LIN {X 0,Y 429.47,Z 573.716,A -85,B 0,C 180,E1 8276.93,E2 8276.93} C_VEL
LIN {X 0,Y 430.465,Z 577.307,A -85,B 0,C 180,E1 8273.605,E2 8273.605} C_VEL
LIN {X 0,Y 428.623,Z 593.36,A -85,B 0,C 180,E1 8273.398,E2 8273.398} C_VEL
LIN {X 0,Y 427.65,Z 601.061,A -85,B 0,C 180,E1 8273.433,E2 8273.433} C_VEL
LIN {X 0,Y 424.746,Z 621.669,A -85,B 0,C 180,E1 8274.011,E2 8274.011} C_VEL
LIN {X 0,Y 423.922,Z 628.276,A -85,B 0,C 180,E1 8274.029,E2 8274.029} C_VEL
LIN {X 0,Y 413.389,Z 717.354,A -85,B 0,C 180,E1 8272.887,E2 8272.887} C_VEL
LIN {X 0,Y 408.118,Z 746.071,A -85,B 0,C 180,E1 8272.482,E2 8272.482} C_VEL
LIN {X 0,Y 402.723,Z 767.743,A -85,B 0,C 180,E1 8272.122,E2 8272.122} C_VEL
LIN {X 0,Y 395.883,Z 790.196,A -85,B 0,C 180,E1 8271.668,E2 8271.668} C_VEL
LIN {X 0,Y 386.127,Z 816.317,A -85,B 0,C 180,E1 8270.974,E2 8270.974} C_VEL
LIN {X 0,Y 377.346,Z 836.309,A -85,B 0,C 180,E1 8270.305,E2 8270.305} C_VEL
LIN {X 0,Y 367.124,Z 856.797,A -85,B 0,C 180,E1 8269.485,E2 8269.485} C_VEL
LIN {X 0,Y 353.895,Z 879.891,A -85,B 0,C 180,E1 8268.336,E2 8268.336} C_VEL
LIN {X 0,Y 341.958,Z 898.335,A -85,B 0,C 180,E1 8267.201,E2 8267.201} C_VEL
LIN {X 0,Y 329.398,Z 915.934,A -85,B 0,C 180,E1 8265.892,E2 8265.892} C_VEL
LIN {X 0,Y 312.582,Z 937.05,A -85,B 0,C 180,E1 8263.94,E2 8263.94} C_VEL
LIN {X 0,Y 298.439,Z 953.025,A -85,B 0,C 180,E1 8262.084,E2 8262.084} C_VEL
LIN {X 0,Y 284.163,Z 967.885,A -85,B 0,C 180,E1 8259.966,E2 8259.966} C_VEL
LIN {X 0,Y 265.558,Z 985.544,A -85,B 0,C 180,E1 8256.739,E2 8256.739} C_VEL
LIN {X 0,Y 250.897,Z 998.283,A -85,B 0,C 180,E1 8253.725,E2 8253.725} C_VEL
LIN {X 0,Y 235.594,Z 1010.758,A -85,B 0,C 180,E1 8249.974,E2 8249.974} C_VEL
LIN {X 0,Y 218.823,Z 1023.439,A -85,B 0,C 180,E1 8244.877,E2 8244.877} C_VEL
LIN {X 0,Y 206.757,Z 1032.129,A -85,B 0,C 180,E1 8240.258,E2 8240.258} C_VEL
LIN {X 0,Y 194.64,Z 1040.684,A -85,B 0,C 180,E1 8234.318,E2 8234.318} C_VEL
LIN {X 0,Y 183.379,Z 1048.53,A -85,B 0,C 180,E1 8226.723,E2 8226.723} C_VEL
LIN {X 0,Y 176.363,Z 1053.655,A -85,B 0,C 180,E1 8219.838,E2 8219.838} C_VEL
LIN {X 0,Y 171.437,Z 1057.709,A -85,B 0,C 180,E1 8212.278,E2 8212.278} C_VEL
LIN {X 0,Y 168.576,Z 1060.697,A -85,B 0,C 180,E1 8203.375,E2 8203.375} C_VEL
LIN {X 0,Y 167.948,Z 1061.835,A -85,B 0,C 180,E1 8196.495,E2 8196.495} C_VEL
LIN {X 0,Y 167.927,Z 1062.025,A -85,B 0,C 180,E1 8190.341,E2 8190.341} C_VEL
LIN {X 0,Y 167.919,Z 1061.465,A -85,B 0,C 180,E1 8184.533,E2 8184.533} C_VEL
LIN {X 0,Y 168.39,Z 1059.828,A -85,B 0,C 180,E1 8177.657,E2 8177.657} C_VEL
LIN {X 0,Y 170.075,Z 1057.173,A -85,B 0,C 180,E1 8170.778,E2 8170.778} C_VEL
LIN {X 0,Y 173.594,Z 1053.274,A -85,B 0,C 180,E1 8163.672,E2 8163.672} C_VEL
LIN {X 0,Y 180.092,Z 1047.442,A -85,B 0,C 180,E1 8155.892,E2 8155.892} C_VEL
LIN {X 0,Y 189.636,Z 1039.498,A -85,B 0,C 180,E1 8148.367,E2 8148.367} C_VEL
LIN {X 0,Y 199.716,Z 1031.446,A -85,B 0,C 180,E1 8142.612,E2 8142.612} C_VEL
LIN {X 0,Y 213.267,Z 1020.629,A -85,B 0,C 180,E1 8136.706,E2 8136.706} C_VEL
LIN {X 0,Y 227.999,Z 1008.192,A -85,B 0,C 180,E1 8131.703,E2 8131.703} C_VEL
LIN {X 0,Y 241.285,Z 996.496,A -85,B 0,C 180,E1 8128.034,E2 8128.034} C_VEL
LIN {X 0,Y 258.503,Z 980.275,A -85,B 0,C 180,E1 8124.099,E2 8124.099} C_VEL
LIN {X 0,Y 272.707,Z 965.724,A -85,B 0,C 180,E1 8121.363,E2 8121.363} C_VEL
LIN {X 0,Y 286.634,Z 950.38,A -85,B 0,C 180,E1 8119.03,E2 8119.03} C_VEL
LIN {X 0,Y 303.56,Z 929.827,A -85,B 0,C 180,E1 8116.562,E2 8116.562} C_VEL
LIN {X 0,Y 316.203,Z 912.825,A -85,B 0,C 180,E1 8114.931,E2 8114.931} C_VEL
LIN {X 0,Y 328.971,Z 893.994,A -85,B 0,C 180,E1 8113.44,E2 8113.44} C_VEL
LIN {X 0,Y 342.461,Z 871.569,A -85,B 0,C 180,E1 8112.014,E2 8112.014} C_VEL
LIN {X 0,Y 352.942,Z 851.881,A -85,B 0,C 180,E1 8110.999,E2 8110.999} C_VEL
LIN {X 0,Y 362.609,Z 831.453,A -85,B 0,C 180,E1 8110.129,E2 8110.129} C_VEL
LIN {X 0,Y 372.867,Z 806.091,A -85,B 0,C 180,E1 8109.259,E2 8109.259} C_VEL
LIN {X 0,Y 380.057,Z 784.957,A -85,B 0,C 180,E1 8108.678,E2 8108.678} C_VEL
LIN {X 0,Y 386.562,Z 762.237,A -85,B 0,C 180,E1 8108.193,E2 8108.193} C_VEL
LIN {X 0,Y 392.552,Z 734.98,A -85,B 0,C 180,E1 8107.729,E2 8107.729} C_VEL
LIN {X 0,Y 396.079,Z 712.548,A -85,B 0,C 180,E1 8107.4,E2 8107.4} C_VEL
LIN {X 0,Y 412.103,Z 569.364,A -85,B 0,C 180,E1 8105.465,E2 8105.465} C_VEL
LIN {X 0,Y 410.53,Z 565.385,A -85,B 0,C 180,E1 8102.513,E2 8102.513} C_VEL
LIN {X 0,Y 409.758,Z 563.185,A -85,B 0,C 180,E1 8098.182,E2 8098.182} C_VEL
LIN {X 0,Y 410.752,Z 565.908,A -85,B 0,C 180,E1 8093.781,E2 8093.781} C_VEL
LIN {X 0,Y 412.109,Z 569.371,A -85,B 0,C 180,E1 8091.348,E2 8091.348} C_VEL
LIN {X 0,Y 395.646,Z 715.398,A -85,B 0,C 180,E1 8089.405,E2 8089.405} C_VEL
LIN {X 0,Y 390.904,Z 742.775,A -85,B 0,C 180,E1 8088.992,E2 8088.992} C_VEL
LIN {X 0,Y 385.342,Z 765.972,A -85,B 0,C 180,E1 8088.555,E2 8088.555} C_VEL
LIN {X 0,Y 379.395,Z 786.292,A -85,B 0,C 180,E1 8088.074,E2 8088.074} C_VEL
LIN {X 0,Y 370.48,Z 811.64,A -85,B 0,C 180,E1 8087.329,E2 8087.329} C_VEL
LIN {X 0,Y 361.399,Z 833.181,A -85,B 0,C 180,E1 8086.531,E2 8086.531} C_VEL
LIN {X 0,Y 351.957,Z 852.896,A -85,B 0,C 180,E1 8085.64,E2 8085.64} C_VEL
LIN {X 0,Y 339.939,Z 875.096,A -85,B 0,C 180,E1 8084.428,E2 8084.428} C_VEL
LIN {X 0,Y 326.959,Z 895.939,A -85,B 0,C 180,E1 8083.014,E2 8083.014} C_VEL
LIN {X 0,Y 314.662,Z 913.816,A -85,B 0,C 180,E1 8081.536,E2 8081.536} C_VEL
LIN {X 0,Y 299.012,Z 934.324,A -85,B 0,C 180,E1 8079.44,E2 8079.44} C_VEL
LIN {X 0,Y 284.739,Z 951.124,A -85,B 0,C 180,E1 8077.277,E2 8077.277} C_VEL
LIN {X 0,Y 270.645,Z 966.445,A -85,B 0,C 180,E1 8074.842,E2 8074.842} C_VEL
LIN {X 0,Y 253.828,Z 983.189,A -85,B 0,C 180,E1 8071.455,E2 8071.455} C_VEL
LIN {X 0,Y 240.068,Z 995.842,A -85,B 0,C 180,E1 8068.175,E2 8068.175} C_VEL
LIN {X 0,Y 226.493,Z 1007.65,A -85,B 0,C 180,E1 8064.32,E2 8064.32} C_VEL
LIN {X 0,Y 210.608,Z 1020.673,A -85,B 0,C 180,E1 8058.706,E2 8058.706} C_VEL
LIN {X 0,Y 199.578,Z 1029.377,A -85,B 0,C 180,E1 8053.739,E2 8053.739} C_VEL
LIN {X 0,Y 189.309,Z 1037.47,A -85,B 0,C 180,E1 8047.784,E2 8047.784} C_VEL
LIN {X 0,Y 179.397,Z 1045.474,A -85,B 0,C 180,E1 8039.739,E2 8039.739} C_VEL
LIN {X 0,Y 173.677,Z 1050.54,A -85,B 0,C 180,E1 8032.689,E2 8032.689} C_VEL
LIN {X 0,Y 170.113,Z 1054.357,A -85,B 0,C 180,E1 8025.428,E2 8025.428} C_VEL
LIN {X 0,Y 168.256,Z 1057.297,A -85,B 0,C 180,E1 8017.053,E2 8017.053} C_VEL
LIN {X 0,Y 167.946,Z 1058.534,A -85,B 0,C 180,E1 8010,E2 8010} C_VEL
LIN {X 0,Y 167.942,Z 1058.789,A -85,B 0,C 180,E1 8003.505,E2 8003.505} C_VEL
LIN {X 0,Y 168.271,Z 1058.165,A -85,B 0,C 180,E1 7996.95,E2 7996.95} C_VEL
LIN {X 0,Y 169.687,Z 1056.537,A -85,B 0,C 180,E1 7990.015,E2 7990.015} C_VEL
LIN {X 0,Y 172.725,Z 1053.867,A -85,B 0,C 180,E1 7983.062,E2 7983.062} C_VEL
LIN {X 0,Y 178.106,Z 1049.841,A -85,B 0,C 180,E1 7975.847,E2 7975.847} C_VEL
LIN {X 0,Y 187.876,Z 1043.071,A -85,B 0,C 180,E1 7967.476,E2 7967.476} C_VEL
LIN {X 0,Y 198.241,Z 1035.985,A -85,B 0,C 180,E1 7961.277,E2 7961.277} C_VEL
LIN {X 0,Y 210.239,Z 1027.705,A -85,B 0,C 180,E1 7955.802,E2 7955.802} C_VEL
LIN {X 0,Y 226.504,Z 1015.937,A -85,B 0,C 180,E1 7950.091,E2 7950.091} C_VEL
LIN {X 0,Y 240.664,Z 1005.04,A -85,B 0,C 180,E1 7946.13,E2 7946.13} C_VEL
LIN {X 0,Y 257.231,Z 991.501,A -85,B 0,C 180,E1 7942.312,E2 7942.312} C_VEL
LIN {X 0,Y 274.025,Z 976.349,A -85,B 0,C 180,E1 7939.081,E2 7939.081} C_VEL
LIN {X 0,Y 288.312,Z 962.437,A -85,B 0,C 180,E1 7936.729,E2 7936.729} C_VEL
LIN {X 0,Y 304.537,Z 945.307,A -85,B 0,C 180,E1 7934.402,E2 7934.402} C_VEL
LIN {X 0,Y 320.435,Z 926.444,A -85,B 0,C 180,E1 7932.397,E2 7932.397} C_VEL
LIN {X 0,Y 333.051,Z 910.04,A -85,B 0,C 180,E1 7930.973,E2 7930.973} C_VEL
LIN {X 0,Y 347.241,Z 889.716,A -85,B 0,C 180,E1 7929.519,E2 7929.519} C_VEL
LIN {X 0,Y 360.273,Z 868.328,A -85,B 0,C 180,E1 7928.298,E2 7928.298} C_VEL
LIN {X 0,Y 370.553,Z 849.453,A -85,B 0,C 180,E1 7927.411,E2 7927.411} C_VEL
LIN {X 0,Y 381.435,Z 826.896,A -85,B 0,C 180,E1 7926.535,E2 7926.535} C_VEL
LIN {X 0,Y 390.957,Z 803.368,A -85,B 0,C 180,E1 7925.801,E2 7925.801} C_VEL
LIN {X 0,Y 398.14,Z 782.602,A -85,B 0,C 180,E1 7925.274,E2 7925.274} C_VEL
LIN {X 0,Y 405.183,Z 758.262,A -85,B 0,C 180,E1 7924.791,E2 7924.791} C_VEL
LIN {X 0,Y 410.782,Z 732.473,A -85,B 0,C 180,E1 7924.388,E2 7924.388} C_VEL
LIN {X 0,Y 414.333,Z 710.195,A -85,B 0,C 180,E1 7924.084,E2 7924.084} C_VEL
LIN {X 0,Y 429.028,Z 584.149,A -85,B 0,C 180,E1 7922.471,E2 7922.471} C_VEL
LIN {X 0,Y 428.424,Z 581.286,A -85,B 0,C 180,E1 7919.465,E2 7919.465} C_VEL
LIN {X 0,Y 428.475,Z 581.6,A -85,B 0,C 180,E1 7917.057,E2 7917.057} C_VEL
LIN {X 0,Y 429.022,Z 584.37,A -85,B 0,C 180,E1 7914.582,E2 7914.582} C_VEL
LIN {X 0,Y 423.922,Z 628.276,A -85,B 0,C 180,E1 7914.029,E2 7914.029} C_VEL
LIN {X 0,Y 422.951,Z 635.978,A -85,B 0,C 180,E1 7914.066,E2 7914.066} C_VEL
LIN {X 0,Y 420.093,Z 656.581,A -85,B 0,C 180,E1 7914.66,E2 7914.66} C_VEL
LIN {X 0,Y 419.271,Z 663.188,A -85,B 0,C 180,E1 7914.678,E2 7914.678} C_VEL
LIN {X 0,Y 412.391,Z 719.368,A -85,B 0,C 180,E1 7913.97,E2 7913.97} C_VEL
LIN {X 0,Y 407.213,Z 746.607,A -85,B 0,C 180,E1 7913.596,E2 7913.596} C_VEL
LIN {X 0,Y 401.82,Z 767.987,A -85,B 0,C 180,E1 7913.256,E2 7913.256} C_VEL
LIN {X 0,Y 394.567,Z 791.474,A -85,B 0,C 180,E1 7912.799,E2 7912.799} C_VEL
LIN {X 0,Y 384.928,Z 816.769,A -85,B 0,C 180,E1 7912.15,E2 7912.15} C_VEL
LIN {X 0,Y 376.077,Z 836.652,A -85,B 0,C 180,E1 7911.512,E2 7911.512} C_VEL
LIN {X 0,Y 365.319,Z 857.898,A -85,B 0,C 180,E1 7910.692,E2 7910.692} C_VEL
LIN {X 0,Y 351.768,Z 881.033,A -85,B 0,C 180,E1 7909.574,E2 7909.574} C_VEL
LIN {X 0,Y 339.795,Z 899.198,A -85,B 0,C 180,E1 7908.49,E2 7908.49} C_VEL
LIN {X 0,Y 325.704,Z 918.528,A -85,B 0,C 180,E1 7907.084,E2 7907.084} C_VEL
LIN {X 0,Y 309.606,Z 938.108,A -85,B 0,C 180,E1 7905.295,E2 7905.295} C_VEL
LIN {X 0,Y 296.015,Z 953.141,A -85,B 0,C 180,E1 7903.597,E2 7903.597} C_VEL
LIN {X 0,Y 280.605,Z 968.825,A -85,B 0,C 180,E1 7901.413,E2 7901.413} C_VEL
LIN {X 0,Y 262.401,Z 985.613,A -85,B 0,C 180,E1 7898.398,E2 7898.398} C_VEL
LIN {X 0,Y 247.337,Z 998.337,A -85,B 0,C 180,E1 7895.448,E2 7895.448} C_VEL
LIN {X 0,Y 230.823,Z 1011.369,A -85,B 0,C 180,E1 7891.565,E2 7891.565} C_VEL
LIN {X 0,Y 214.145,Z 1023.454,A -85,B 0,C 180,E1 7886.698,E2 7886.698} C_VEL
LIN {X 0,Y 201.29,Z 1032.299,A -85,B 0,C 180,E1 7881.978,E2 7881.978} C_VEL
LIN {X 0,Y 187.765,Z 1041.384,A -85,B 0,C 180,E1 7875.527,E2 7875.527} C_VEL
LIN {X 0,Y 176.383,Z 1048.771,A -85,B 0,C 180,E1 7868.003,E2 7868.003} C_VEL
LIN {X 0,Y 169.025,Z 1053.775,A -85,B 0,C 180,E1 7860.975,E2 7860.975} C_VEL
LIN {X 0,Y 163.349,Z 1058.145,A -85,B 0,C 180,E1 7852.304,E2 7852.304} C_VEL
LIN {X 0,Y 160.616,Z 1060.701,A -85,B 0,C 180,E1 7843.684,E2 7843.684} C_VEL
LIN {X 0,Y 159.96,Z 1061.761,A -85,B 0,C 180,E1 7836.821,E2 7836.821} C_VEL
LIN {X 0,Y 159.919,Z 1061.965,A -85,B 0,C 180,E1 7830.717,E2 7830.717} C_VEL
LIN {X 0,Y 159.918,Z 1061.442,A -85,B 0,C 180,E1 7824.619,E2 7824.619} C_VEL
LIN {X 0,Y 160.417,Z 1059.841,A -85,B 0,C 180,E1 7817.399,E2 7817.399} C_VEL
LIN {X 0,Y 162.361,Z 1057.061,A -85,B 0,C 180,E1 7809.826,E2 7809.826} C_VEL
LIN {X 0,Y 166.24,Z 1053.152,A -85,B 0,C 180,E1 7802.411,E2 7802.411} C_VEL
LIN {X 0,Y 173.632,Z 1047.046,A -85,B 0,C 180,E1 7794.029,E2 7794.029} C_VEL
LIN {X 0,Y 183.953,Z 1038.984,A -85,B 0,C 180,E1 7786.345,E2 7786.345} C_VEL
LIN {X 0,Y 194.712,Z 1030.869,A -85,B 0,C 180,E1 7780.535,E2 7780.535} C_VEL
LIN {X 0,Y 209.647,Z 1019.395,A -85,B 0,C 180,E1 7774.401,E2 7774.401} C_VEL
LIN {X 0,Y 223.722,Z 1007.99,A -85,B 0,C 180,E1 7769.883,E2 7769.883} C_VEL
LIN {X 0,Y 238.228,Z 995.638,A -85,B 0,C 180,E1 7766.078,E2 7766.078} C_VEL
LIN {X 0,Y 256.005,Z 979.251,A -85,B 0,C 180,E1 7762.233,E2 7762.233} C_VEL
LIN {X 0,Y 269.87,Z 965.379,A -85,B 0,C 180,E1 7759.704,E2 7759.704} C_VEL
LIN {X 0,Y 284.039,Z 950.103,A -85,B 0,C 180,E1 7757.45,E2 7757.45} C_VEL
LIN {X 0,Y 300.811,Z 930.15,A -85,B 0,C 180,E1 7755.12,E2 7755.12} C_VEL
LIN {X 0,Y 313.679,Z 913.18,A -85,B 0,C 180,E1 7753.538,E2 7753.538} C_VEL
LIN {X 0,Y 326.253,Z 894.982,A -85,B 0,C 180,E1 7752.135,E2 7752.135} C_VEL
LIN {X 0,Y 340.851,Z 871.148,A -85,B 0,C 180,E1 7750.667,E2 7750.667} C_VEL
LIN {X 0,Y 351.011,Z 852.333,A -85,B 0,C 180,E1 7749.732,E2 7749.732} C_VEL
LIN {X 0,Y 360.329,Z 832.982,A -85,B 0,C 180,E1 7748.933,E2 7748.933} C_VEL
LIN {X 0,Y 370.654,Z 808.205,A -85,B 0,C 180,E1 7748.099,E2 7748.099} C_VEL
LIN {X 0,Y 378.444,Z 785.754,A -85,B 0,C 180,E1 7747.5,E2 7747.5} C_VEL
LIN {X 0,Y 384.802,Z 763.973,A -85,B 0,C 180,E1 7747.05,E2 7747.05} C_VEL
LIN {X 0,Y 391.137,Z 736.073,A -85,B 0,C 180,E1 7746.587,E2 7746.587} C_VEL
LIN {X 0,Y 394.832,Z 713.123,A -85,B 0,C 180,E1 7746.258,E2 7746.258} C_VEL
LIN {X 0,Y 410.46,Z 575.932,A -85,B 0,C 180,E1 7744.453,E2 7744.453} C_VEL
LIN {X 0,Y 409.492,Z 573.267,A -85,B 0,C 180,E1 7742.379,E2 7742.379} C_VEL
LIN {X 0,Y 408.781,Z 571.142,A -85,B 0,C 180,E1 7738.178,E2 7738.178} C_VEL
LIN {X 0,Y 409.707,Z 573.818,A -85,B 0,C 180,E1 7733.906,E2 7733.906} C_VEL
LIN {X 0,Y 410.429,Z 576.164,A -85,B 0,C 180,E1 7732.37,E2 7732.37} C_VEL
LIN {X 0,Y 394.459,Z 715.538,A -85,B 0,C 180,E1 7730.554,E2 7730.554} C_VEL
LIN {X 0,Y 389.648,Z 742.945,A -85,B 0,C 180,E1 7730.153,E2 7730.153} C_VEL
LIN {X 0,Y 384.031,Z 766.109,A -85,B 0,C 180,E1 7729.733,E2 7729.733} C_VEL
LIN {X 0,Y 378.06,Z 786.281,A -85,B 0,C 180,E1 7729.275,E2 7729.275} C_VEL
LIN {X 0,Y 369.271,Z 811.091,A -85,B 0,C 180,E1 7728.578,E2 7728.578} C_VEL
LIN {X 0,Y 359.619,Z 833.698,A -85,B 0,C 180,E1 7727.771,E2 7727.771} C_VEL
LIN {X 0,Y 350.054,Z 853.368,A -85,B 0,C 180,E1 7726.911,E2 7726.911} C_VEL
LIN {X 0,Y 337.418,Z 876.224,A -85,B 0,C 180,E1 7725.698,E2 7725.698} C_VEL
LIN {X 0,Y 324.93,Z 895.957,A -85,B 0,C 180,E1 7724.401,E2 7724.401} C_VEL
LIN {X 0,Y 312.63,Z 913.561,A -85,B 0,C 180,E1 7722.997,E2 7722.997} C_VEL
LIN {X 0,Y 297.114,Z 933.624,A -85,B 0,C 180,E1 7721.024,E2 7721.024} C_VEL
LIN {X 0,Y 282.804,Z 950.19,A -85,B 0,C 180,E1 7718.971,E2 7718.971} C_VEL
LIN {X 0,Y 268.893,Z 965.042,A -85,B 0,C 180,E1 7716.704,E2 7716.704} C_VEL
LIN {X 0,Y 252.334,Z 981.35,A -85,B 0,C 180,E1 7713.577,E2 7713.577} C_VEL
LIN {X 0,Y 236.579,Z 995.438,A -85,B 0,C 180,E1 7710.045,E2 7710.045} C_VEL
LIN {X 0,Y 223.168,Z 1006.728,A -85,B 0,C 180,E1 7706.445,E2 7706.445} C_VEL
LIN {X 0,Y 207.578,Z 1019.163,A -85,B 0,C 180,E1 7701.291,E2 7701.291} C_VEL
LIN {X 0,Y 194.274,Z 1029.15,A -85,B 0,C 180,E1 7695.676,E2 7695.676} C_VEL
LIN {X 0,Y 183.355,Z 1037.283,A -85,B 0,C 180,E1 7689.645,E2 7689.645} C_VEL
LIN {X 0,Y 172.691,Z 1045.361,A -85,B 0,C 180,E1 7681.406,E2 7681.406} C_VEL
LIN {X 0,Y 166.346,Z 1050.539,A -85,B 0,C 180,E1 7673.984,E2 7673.984} C_VEL
LIN {X 0,Y 162.43,Z 1054.356,A -85,B 0,C 180,E1 7666.449,E2 7666.449} C_VEL
LIN {X 0,Y 160.346,Z 1057.294,A -85,B 0,C 180,E1 7657.885,E2 7657.885} C_VEL
LIN {X 0,Y 159.951,Z 1058.594,A -85,B 0,C 180,E1 7650.358,E2 7650.358} C_VEL
LIN {X 0,Y 159.939,Z 1058.896,A -85,B 0,C 180,E1 7643.735,E2 7643.735} C_VEL
LIN {X 0,Y 160.298,Z 1058.296,A -85,B 0,C 180,E1 7636.656,E2 7636.656} C_VEL
LIN {X 0,Y 161.961,Z 1056.591,A -85,B 0,C 180,E1 7629.018,E2 7629.018} C_VEL
LIN {X 0,Y 165.3,Z 1053.952,A -85,B 0,C 180,E1 7621.848,E2 7621.848} C_VEL
LIN {X 0,Y 170.916,Z 1050.08,A -85,B 0,C 180,E1 7614.608,E2 7614.608} C_VEL
LIN {X 0,Y 180.863,Z 1043.688,A -85,B 0,C 180,E1 7606.287,E2 7606.287} C_VEL
LIN {X 0,Y 192.233,Z 1036.337,A -85,B 0,C 180,E1 7599.663,E2 7599.663} C_VEL
LIN {X 0,Y 204.649,Z 1028.189,A -85,B 0,C 180,E1 7594.186,E2 7594.186} C_VEL
LIN {X 0,Y 221.691,Z 1016.415,A -85,B 0,C 180,E1 7588.418,E2 7588.418} C_VEL
LIN {X 0,Y 236.248,Z 1005.617,A -85,B 0,C 180,E1 7584.501,E2 7584.501} C_VEL
LIN {X 0,Y 250.963,Z 993.989,A -85,B 0,C 180,E1 7581.204,E2 7581.204} C_VEL
LIN {X 0,Y 269.727,Z 977.804,A -85,B 0,C 180,E1 7577.692,E2 7577.692} C_VEL
LIN {X 0,Y 284.17,Z 964.146,A -85,B 0,C 180,E1 7575.399,E2 7575.399} C_VEL
LIN {X 0,Y 299.025,Z 948.913,A -85,B 0,C 180,E1 7573.332,E2 7573.332} C_VEL
LIN {X 0,Y 316.3,Z 929.304,A -85,B 0,C 180,E1 7571.221,E2 7571.221} C_VEL
LIN {X 0,Y 329.734,Z 912.297,A -85,B 0,C 180,E1 7569.759,E2 7569.759} C_VEL
LIN {X 0,Y 342.234,Z 894.891,A -85,B 0,C 180,E1 7568.516,E2 7568.516} C_VEL
LIN {X 0,Y 356.78,Z 872.204,A -85,B 0,C 180,E1 7567.209,E2 7567.209} C_VEL
LIN {X 0,Y 368.158,Z 851.855,A -85,B 0,C 180,E1 7566.267,E2 7566.267} C_VEL
LIN {X 0,Y 377.711,Z 832.613,A -85,B 0,C 180,E1 7565.524,E2 7565.524} C_VEL
LIN {X 0,Y 388.288,Z 808.07,A -85,B 0,C 180,E1 7564.749,E2 7564.749} C_VEL
LIN {X 0,Y 396.506,Z 785.025,A -85,B 0,C 180,E1 7564.175,E2 7564.175} C_VEL
LIN {X 0,Y 402.699,Z 764.375,A -85,B 0,C 180,E1 7563.767,E2 7563.767} C_VEL
LIN {X 0,Y 408.913,Z 738.596,A -85,B 0,C 180,E1 7563.356,E2 7563.356} C_VEL
LIN {X 0,Y 413.167,Z 713.559,A -85,B 0,C 180,E1 7563.021,E2 7563.021} C_VEL
LIN {X 0,Y 427.715,Z 591.178,A -85,B 0,C 180,E1 7561.474,E2 7561.474} C_VEL
LIN {X 0,Y 427.448,Z 589.227,A -85,B 0,C 180,E1 7559.464,E2 7559.464} C_VEL
LIN {X 0,Y 427.485,Z 589.541,A -85,B 0,C 180,E1 7557.135,E2 7557.135} C_VEL
LIN {X 0,Y 427.714,Z 591.357,A -85,B 0,C 180,E1 7555.567,E2 7555.567} C_VEL
LIN {X 0,Y 419.271,Z 663.188,A -85,B 0,C 180,E1 7554.678,E2 7554.678} C_VEL
LIN {X 0,Y 418.304,Z 670.889,A -85,B 0,C 180,E1 7554.717,E2 7554.717} C_VEL
LIN {X 0,Y 415.494,Z 691.484,A -85,B 0,C 180,E1 7555.328,E2 7555.328} C_VEL
LIN {X 0,Y 414.674,Z 698.09,A -85,B 0,C 180,E1 7555.348,E2 7555.348} C_VEL
LIN {X 0,Y 410.27,Z 728.43,A -85,B 0,C 180,E1 7554.967,E2 7554.967} C_VEL
LIN {X 0,Y 405.642,Z 750.656,A -85,B 0,C 180,E1 7554.667,E2 7554.667} C_VEL
LIN {X 0,Y 399.101,Z 775.285,A -85,B 0,C 180,E1 7554.274,E2 7554.274} C_VEL
LIN {X 0,Y 390.762,Z 799.859,A -85,B 0,C 180,E1 7553.771,E2 7553.771} C_VEL
LIN {X 0,Y 382.541,Z 820.389,A -85,B 0,C 180,E1 7553.245,E2 7553.245} C_VEL
LIN {X 0,Y 371.547,Z 844.159,A -85,B 0,C 180,E1 7552.483,E2 7552.483} C_VEL
LIN {X 0,Y 359.498,Z 866.24,A -85,B 0,C 180,E1 7551.592,E2 7551.592} C_VEL
LIN {X 0,Y 348.522,Z 884.184,A -85,B 0,C 180,E1 7550.72,E2 7550.72} C_VEL
LIN {X 0,Y 334.103,Z 905.369,A -85,B 0,C 180,E1 7549.457,E2 7549.457} C_VEL
LIN {X 0,Y 318.639,Z 925.256,A -85,B 0,C 180,E1 7547.956,E2 7547.956} C_VEL
LIN {X 0,Y 304.935,Z 941.267,A -85,B 0,C 180,E1 7546.465,E2 7546.465} C_VEL
LIN {X 0,Y 288.531,Z 958.784,A -85,B 0,C 180,E1 7544.448,E2 7544.448} C_VEL
LIN {X 0,Y 271.243,Z 975.26,A -85,B 0,C 180,E1 7542.002,E2 7542.002} C_VEL
LIN {X 0,Y 256.167,Z 988.472,A -85,B 0,C 180,E1 7539.518,E2 7539.518} C_VEL
LIN {X 0,Y 238.49,Z 1002.819,A -85,B 0,C 180,E1 7536.061,E2 7536.061} C_VEL
LIN {X 0,Y 221.05,Z 1015.595,A -85,B 0,C 180,E1 7531.891,E2 7531.891} C_VEL
LIN {X 0,Y 206.959,Z 1025.303,A -85,B 0,C 180,E1 7527.724,E2 7527.724} C_VEL
LIN {X 0,Y 191.052,Z 1035.72,A -85,B 0,C 180,E1 7521.724,E2 7521.724} C_VEL
LIN {X 0,Y 177.894,Z 1043.82,A -85,B 0,C 180,E1 7515.089,E2 7515.089} C_VEL
LIN {X 0,Y 168.032,Z 1049.921,A -85,B 0,C 180,E1 7508.233,E2 7508.233} C_VEL
LIN {X 0,Y 159.124,Z 1055.678,A -85,B 0,C 180,E1 7498.937,E2 7498.937} C_VEL
LIN {X 0,Y 154.472,Z 1059.035,A -85,B 0,C 180,E1 7490.459,E2 7490.459} C_VEL
LIN {X 0,Y 152.467,Z 1060.914,A -85,B 0,C 180,E1 7482.884,E2 7482.884} C_VEL
LIN {X 0,Y 151.944,Z 1061.735,A -85,B 0,C 180,E1 7476.423,E2 7476.423} C_VEL
LIN {X 0,Y 151.926,Z 1061.86,A -85,B 0,C 180,E1 7470.377,E2 7470.377} C_VEL
LIN {X 0,Y 151.932,Z 1061.281,A -85,B 0,C 180,E1 7463.956,E2 7463.956} C_VEL
LIN {X 0,Y 152.568,Z 1059.624,A -85,B 0,C 180,E1 7456.354,E2 7456.354} C_VEL
LIN {X 0,Y 154.693,Z 1056.949,A -85,B 0,C 180,E1 7448.779,E2 7448.779} C_VEL
LIN {X 0,Y 158.966,Z 1053.029,A -85,B 0,C 180,E1 7441.032,E2 7441.032} C_VEL
LIN {X 0,Y 166.981,Z 1046.908,A -85,B 0,C 180,E1 7432.354,E2 7432.354} C_VEL
LIN {X 0,Y 177.634,Z 1039.103,A -85,B 0,C 180,E1 7424.718,E2 7424.718} C_VEL
LIN {X 0,Y 188.806,Z 1031.113,A -85,B 0,C 180,E1 7418.878,E2 7418.878} C_VEL
LIN {X 0,Y 203.714,Z 1020.249,A -85,B 0,C 180,E1 7412.932,E2 7412.932} C_VEL
LIN {X 0,Y 218.955,Z 1008.369,A -85,B 0,C 180,E1 7408.194,E2 7408.194} C_VEL
LIN {X 0,Y 233.284,Z 996.587,A -85,B 0,C 180,E1 7404.567,E2 7404.567} C_VEL
LIN {X 0,Y 250.533,Z 981.346,A -85,B 0,C 180,E1 7400.949,E2 7400.949} C_VEL
LIN {X 0,Y 266.412,Z 965.899,A -85,B 0,C 180,E1 7398.151,E2 7398.151} C_VEL
LIN {X 0,Y 279.93,Z 951.698,A -85,B 0,C 180,E1 7396.087,E2 7396.087} C_VEL
LIN {X 0,Y 296.158,Z 933.126,A -85,B 0,C 180,E1 7393.916,E2 7393.916} C_VEL
LIN {X 0,Y 310.948,Z 914.072,A -85,B 0,C 180,E1 7392.166,E2 7392.166} C_VEL
LIN {X 0,Y 323.201,Z 896.712,A -85,B 0,C 180,E1 7390.86,E2 7390.86} C_VEL
LIN {X 0,Y 337.106,Z 874.825,A -85,B 0,C 180,E1 7389.522,E2 7389.522} C_VEL
LIN {X 0,Y 349.252,Z 852.784,A -85,B 0,C 180,E1 7388.452,E2 7388.452} C_VEL
LIN {X 0,Y 358.607,Z 833.652,A -85,B 0,C 180,E1 7387.691,E2 7387.691} C_VEL
LIN {X 0,Y 368.644,Z 810.182,A -85,B 0,C 180,E1 7386.923,E2 7386.923} C_VEL
LIN {X 0,Y 376.95,Z 786.68,A -85,B 0,C 180,E1 7386.316,E2 7386.316} C_VEL
LIN {X 0,Y 383.291,Z 765.353,A -85,B 0,C 180,E1 7385.89,E2 7385.89} C_VEL
LIN {X 0,Y 389.416,Z 739.696,A -85,B 0,C 180,E1 7385.472,E2 7385.472} C_VEL
LIN {X 0,Y 393.635,Z 714.463,A -85,B 0,C 180,E1 7385.12,E2 7385.12} C_VEL
LIN {X 0,Y 408.929,Z 582.638,A -85,B 0,C 180,E1 7383.434,E2 7383.434} C_VEL
LIN {X 0,Y 408.402,Z 581.066,A -85,B 0,C 180,E1 7382.105,E2 7382.105} C_VEL
LIN {X 0,Y 407.803,Z 579.102,A -85,B 0,C 180,E1 7378.173,E2 7378.173} C_VEL
LIN {X 0,Y 408.638,Z 581.623,A -85,B 0,C 180,E1 7374.101,E2 7374.101} C_VEL
LIN {X 0,Y 408.894,Z 582.831,A -85,B 0,C 180,E1 7373.402,E2 7373.402} C_VEL
LIN {X 0,Y 393.425,Z 715.701,A -85,B 0,C 180,E1 7371.709,E2 7371.709} C_VEL
LIN {X 0,Y 388.5,Z 743.337,A -85,B 0,C 180,E1 7371.318,E2 7371.318} C_VEL
LIN {X 0,Y 382.85,Z 766.362,A -85,B 0,C 180,E1 7370.917,E2 7370.917} C_VEL
LIN {X 0,Y 376.658,Z 787.001,A -85,B 0,C 180,E1 7370.466,E2 7370.466} C_VEL
LIN {X 0,Y 367.306,Z 812.781,A -85,B 0,C 180,E1 7369.762,E2 7369.762} C_VEL
LIN {X 0,Y 358.01,Z 834.214,A -85,B 0,C 180,E1 7369.022,E2 7369.022} C_VEL
LIN {X 0,Y 348.326,Z 853.839,A -85,B 0,C 180,E1 7368.196,E2 7368.196} C_VEL
LIN {X 0,Y 335.066,Z 877.352,A -85,B 0,C 180,E1 7366.987,E2 7366.987} C_VEL
LIN {X 0,Y 322.854,Z 896.329,A -85,B 0,C 180,E1 7365.781,E2 7365.781} C_VEL
LIN {X 0,Y 310.363,Z 913.908,A -85,B 0,C 180,E1 7364.424,E2 7364.424} C_VEL
LIN {X 0,Y 294.142,Z 934.428,A -85,B 0,C 180,E1 7362.46,E2 7362.46} C_VEL
LIN {X 0,Y 279.142,Z 951.39,A -85,B 0,C 180,E1 7360.401,E2 7360.401} C_VEL
LIN {X 0,Y 264.953,Z 966.144,A -85,B 0,C 180,E1 7358.18,E2 7358.18} C_VEL
LIN {X 0,Y 246.31,Z 983.773,A -85,B 0,C 180,E1 7354.77,E2 7354.77} C_VEL
LIN {X 0,Y 231.85,Z 996.288,A -85,B 0,C 180,E1 7351.615,E2 7351.615} C_VEL
LIN {X 0,Y 216.614,Z 1008.654,A -85,B 0,C 180,E1 7347.625,E2 7347.625} C_VEL
LIN {X 0,Y 200.636,Z 1020.704,A -85,B 0,C 180,E1 7342.409,E2 7342.409} C_VEL
LIN {X 0,Y 188.072,Z 1029.721,A -85,B 0,C 180,E1 7337.195,E2 7337.195} C_VEL
LIN {X 0,Y 176.176,Z 1038.139,A -85,B 0,C 180,E1 7330.744,E2 7330.744} C_VEL
LIN {X 0,Y 165.416,Z 1045.749,A -85,B 0,C 180,E1 7322.546,E2 7322.546} C_VEL
LIN {X 0,Y 159.041,Z 1050.589,A -85,B 0,C 180,E1 7315.31,E2 7315.31} C_VEL
LIN {X 0,Y 154.832,Z 1054.314,A -85,B 0,C 180,E1 7307.669,E2 7307.669} C_VEL
LIN {X 0,Y 152.495,Z 1057.178,A -85,B 0,C 180,E1 7299.054,E2 7299.054} C_VEL
LIN {X 0,Y 151.946,Z 1058.633,A -85,B 0,C 180,E1 7291.131,E2 7291.131} C_VEL
LIN {X 0,Y 151.928,Z 1059.023,A -85,B 0,C 180,E1 7284.334,E2 7284.334} C_VEL
LIN {X 0,Y 152.288,Z 1058.493,A -85,B 0,C 180,E1 7276.714,E2 7276.714} C_VEL
LIN {X 0,Y 154.149,Z 1056.758,A -85,B 0,C 180,E1 7268.301,E2 7268.301} C_VEL
LIN {X 0,Y 158.014,Z 1053.996,A -85,B 0,C 180,E1 7260.424,E2 7260.424} C_VEL
LIN {X 0,Y 164.506,Z 1049.908,A -85,B 0,C 180,E1 7252.569,E2 7252.569} C_VEL
LIN {X 0,Y 175.831,Z 1043.093,A -85,B 0,C 180,E1 7243.763,E2 7243.763} C_VEL
LIN {X 0,Y 187.528,Z 1035.984,A -85,B 0,C 180,E1 7237.396,E2 7237.396} C_VEL
LIN {X 0,Y 201.139,Z 1027.49,A -85,B 0,C 180,E1 7231.782,E2 7231.782} C_VEL
LIN {X 0,Y 218.529,Z 1015.861,A -85,B 0,C 180,E1 7226.259,E2 7226.259} C_VEL
LIN {X 0,Y 232.878,Z 1005.568,A -85,B 0,C 180,E1 7222.613,E2 7222.613} C_VEL
LIN {X 0,Y 248.862,Z 993.287,A -85,B 0,C 180,E1 7219.232,E2 7219.232} C_VEL
LIN {X 0,Y 267.299,Z 977.71,A -85,B 0,C 180,E1 7215.98,E2 7215.98} C_VEL
LIN {X 0,Y 282.305,Z 963.803,A -85,B 0,C 180,E1 7213.728,E2 7213.728} C_VEL
LIN {X 0,Y 297.5,Z 948.487,A -85,B 0,C 180,E1 7211.732,E2 7211.732} C_VEL
LIN {X 0,Y 315.445,Z 928.34,A -85,B 0,C 180,E1 7209.668,E2 7209.668} C_VEL
LIN {X 0,Y 328.902,Z 911.491,A -85,B 0,C 180,E1 7208.293,E2 7208.293} C_VEL
LIN {X 0,Y 342.26,Z 893.04,A -85,B 0,C 180,E1 7207.048,E2 7207.048} C_VEL
LIN {X 0,Y 356.798,Z 870.289,A -85,B 0,C 180,E1 7205.819,E2 7205.819} C_VEL
LIN {X 0,Y 367.835,Z 850.633,A -85,B 0,C 180,E1 7204.96,E2 7204.96} C_VEL
LIN {X 0,Y 377.983,Z 830.228,A -85,B 0,C 180,E1 7204.223,E2 7204.223} C_VEL
LIN {X 0,Y 388.674,Z 804.999,A -85,B 0,C 180,E1 7203.486,E2 7203.486} C_VEL
LIN {X 0,Y 396.118,Z 784.091,A -85,B 0,C 180,E1 7202.994,E2 7202.994} C_VEL
LIN {X 0,Y 402.607,Z 762.421,A -85,B 0,C 180,E1 7202.593,E2 7202.593} C_VEL
LIN {X 0,Y 409.092,Z 734.475,A -85,B 0,C 180,E1 7202.179,E2 7202.179} C_VEL
LIN {X 0,Y 412.849,Z 711.925,A -85,B 0,C 180,E1 7201.89,E2 7201.89} C_VEL
LIN {X 0,Y 426.546,Z 598.162,A -85,B 0,C 180,E1 7200.504,E2 7200.504} C_VEL
LIN {X 0,Y 426.458,Z 597.165,A -85,B 0,C 180,E1 7199.328,E2 7199.328} C_VEL
LIN {X 0,Y 426.497,Z 597.52,A -85,B 0,C 180,E1 7197.178,E2 7197.178} C_VEL
LIN {X 0,Y 426.517,Z 598.471,A -85,B 0,C 180,E1 7196.556,E2 7196.556} C_VEL
LIN {X 0,Y 414.674,Z 698.09,A -85,B 0,C 180,E1 7195.348,E2 7195.348} C_VEL
LIN {X 0,Y 413.682,Z 705.782,A -85,B 0,C 180,E1 7195.388,E2 7195.388} C_VEL
LIN {X 0,Y 410.299,Z 726.277,A -85,B 0,C 180,E1 7196.018,E2 7196.018} C_VEL
LIN {X 0,Y 409.011,Z 732.823,A -85,B 0,C 180,E1 7196.031,E2 7196.031} C_VEL
LIN {X 0,Y 403.22,Z 758.819,A -85,B 0,C 180,E1 7195.688,E2 7195.688} C_VEL
LIN {X 0,Y 395.816,Z 783.689,A -85,B 0,C 180,E1 7195.281,E2 7195.281} C_VEL
LIN {X 0,Y 389.007,Z 802.871,A -85,B 0,C 180,E1 7194.88,E2 7194.88} C_VEL
LIN {X 0,Y 379.339,Z 826.239,A -85,B 0,C 180,E1 7194.289,E2 7194.289} C_VEL
LIN {X 0,Y 367.797,Z 849.648,A -85,B 0,C 180,E1 7193.535,E2 7193.535} C_VEL
LIN {X 0,Y 356.888,Z 869.076,A -85,B 0,C 180,E1 7192.757,E2 7192.757} C_VEL
LIN {X 0,Y 343.533,Z 890.257,A -85,B 0,C 180,E1 7191.73,E2 7191.73} C_VEL
LIN {X 0,Y 328.501,Z 911.02,A -85,B 0,C 180,E1 7190.465,E2 7190.465} C_VEL
LIN {X 0,Y 315.113,Z 927.71,A -85,B 0,C 180,E1 7189.21,E2 7189.21} C_VEL
LIN {X 0,Y 298.581,Z 946.44,A -85,B 0,C 180,E1 7187.467,E2 7187.467} C_VEL
LIN {X 0,Y 281.093,Z 963.973,A -85,B 0,C 180,E1 7185.362,E2 7185.362} C_VEL
LIN {X 0,Y 265.344,Z 978.412,A -85,B 0,C 180,E1 7183.164,E2 7183.164} C_VEL
LIN {X 0,Y 246.605,Z 994.087,A -85,B 0,C 180,E1 7180.087,E2 7180.087} C_VEL
LIN {X 0,Y 229.647,Z 1006.878,A -85,B 0,C 180,E1 7176.736,E2 7176.736} C_VEL
LIN {X 0,Y 214.251,Z 1017.679,A -85,B 0,C 180,E1 7173.047,E2 7173.047} C_VEL
LIN {X 0,Y 196.426,Z 1029.306,A -85,B 0,C 180,E1 7167.673,E2 7167.673} C_VEL
LIN {X 0,Y 181.723,Z 1038.188,A -85,B 0,C 180,E1 7161.89,E2 7161.89} C_VEL
LIN {X 0,Y 169.539,Z 1045.321,A -85,B 0,C 180,E1 7155.53,E2 7155.53} C_VEL
LIN {X 0,Y 157.212,Z 1052.451,A -85,B 0,C 180,E1 7146.263,E2 7146.263} C_VEL
LIN {X 0,Y 150.339,Z 1056.599,A -85,B 0,C 180,E1 7138.178,E2 7138.178} C_VEL
LIN {X 0,Y 146.222,Z 1059.44,A -85,B 0,C 180,E1 7129.993,E2 7129.993} C_VEL
LIN {X 0,Y 144.197,Z 1061.336,A -85,B 0,C 180,E1 7120.791,E2 7120.791} C_VEL
LIN {X 0,Y 143.907,Z 1061.874,A -85,B 0,C 180,E1 7113.187,E2 7113.187} C_VEL
LIN {X 0,Y 143.909,Z 1061.596,A -85,B 0,C 180,E1 7107.212,E2 7107.212} C_VEL
LIN {X 0,Y 144.117,Z 1060.566,A -85,B 0,C 180,E1 7100.012,E2 7100.012} C_VEL
LIN {X 0,Y 146.023,Z 1057.974,A -85,B 0,C 180,E1 7090.396,E2 7090.396} C_VEL
LIN {X 0,Y 150.71,Z 1053.747,A -85,B 0,C 180,E1 7081.033,E2 7081.033} C_VEL
LIN {X 0,Y 157.343,Z 1048.851,A -85,B 0,C 180,E1 7073.32,E2 7073.32} C_VEL
LIN {X 0,Y 167.986,Z 1041.658,A -85,B 0,C 180,E1 7065.098,E2 7065.098} C_VEL
LIN {X 0,Y 181.272,Z 1032.59,A -85,B 0,C 180,E1 7057.929,E2 7057.929} C_VEL
LIN {X 0,Y 193.888,Z 1023.834,A -85,B 0,C 180,E1 7052.785,E2 7052.785} C_VEL
LIN {X 0,Y 209.952,Z 1012.224,A -85,B 0,C 180,E1 7047.649,E2 7047.649} C_VEL
LIN {X 0,Y 226.777,Z 998.949,A -85,B 0,C 180,E1 7043.38,E2 7043.38} C_VEL
LIN {X 0,Y 241.066,Z 986.905,A -85,B 0,C 180,E1 7040.382,E2 7040.382} C_VEL
LIN {X 0,Y 258.643,Z 970.931,A -85,B 0,C 180,E1 7037.279,E2 7037.279} C_VEL
LIN {X 0,Y 275.103,Z 954.231,A -85,B 0,C 180,E1 7034.806,E2 7034.806} C_VEL
LIN {X 0,Y 288.842,Z 939.07,A -85,B 0,C 180,E1 7033.004,E2 7033.004} C_VEL
LIN {X 0,Y 304.779,Z 919.821,A -85,B 0,C 180,E1 7031.161,E2 7031.161} C_VEL
LIN {X 0,Y 319.476,Z 899.657,A -85,B 0,C 180,E1 7029.642,E2 7029.642} C_VEL
LIN {X 0,Y 331.617,Z 881.217,A -85,B 0,C 180,E1 7028.515,E2 7028.515} C_VEL
LIN {X 0,Y 344.829,Z 858.692,A -85,B 0,C 180,E1 7027.396,E2 7027.396} C_VEL
LIN {X 0,Y 355.614,Z 837.382,A -85,B 0,C 180,E1 7026.545,E2 7026.545} C_VEL
LIN {X 0,Y 364.385,Z 817.685,A -85,B 0,C 180,E1 7025.896,E2 7025.896} C_VEL
LIN {X 0,Y 373.776,Z 793.304,A -85,B 0,C 180,E1 7025.253,E2 7025.253} C_VEL
LIN {X 0,Y 381.38,Z 768.746,A -85,B 0,C 180,E1 7024.758,E2 7024.758} C_VEL
LIN {X 0,Y 386.794,Z 747.309,A -85,B 0,C 180,E1 7024.409,E2 7024.409} C_VEL
LIN {X 0,Y 391.912,Z 720.747,A -85,B 0,C 180,E1 7024.039,E2 7024.039} C_VEL
LIN {X 0,Y 398.092,Z 670.37,A -85,B 0,C 180,E1 7023.402,E2 7023.402} C_VEL
LIN {X 0,Y 407.531,Z 589.243,A -85,B 0,C 180,E1 7022.391,E2 7022.391} C_VEL
LIN {X 0,Y 406.826,Z 587.063,A -85,B 0,C 180,E1 7018.169,E2 7018.169} C_VEL
LIN {X 0,Y 407.515,Z 589.313,A -85,B 0,C 180,E1 7014.445,E2 7014.445} C_VEL
LIN {X 0,Y 392.552,Z 715.858,A -85,B 0,C 180,E1 7012.87,E2 7012.87} C_VEL
LIN {X 0,Y 387.559,Z 743.527,A -85,B 0,C 180,E1 7012.492,E2 7012.492} C_VEL
LIN {X 0,Y 381.853,Z 766.534,A -85,B 0,C 180,E1 7012.108,E2 7012.108} C_VEL
LIN {X 0,Y 375.656,Z 786.978,A -85,B 0,C 180,E1 7011.684,E2 7011.684} C_VEL
LIN {X 0,Y 366.441,Z 812.226,A -85,B 0,C 180,E1 7011.028,E2 7011.028} C_VEL
LIN {X 0,Y 357.042,Z 833.733,A -85,B 0,C 180,E1 7010.32,E2 7010.32} C_VEL
LIN {X 0,Y 347.286,Z 853.331,A -85,B 0,C 180,E1 7009.535,E2 7009.535} C_VEL
LIN {X 0,Y 334.269,Z 876.297,A -85,B 0,C 180,E1 7008.417,E2 7008.417} C_VEL
LIN {X 0,Y 321.424,Z 896.04,A -85,B 0,C 180,E1 7007.222,E2 7007.222} C_VEL
LIN {X 0,Y 308.786,Z 913.592,A -85,B 0,C 180,E1 7005.924,E2 7005.924} C_VEL
LIN {X 0,Y 292.687,Z 933.728,A -85,B 0,C 180,E1 7004.084,E2 7004.084} C_VEL
LIN {X 0,Y 277.388,Z 950.758,A -85,B 0,C 180,E1 7002.106,E2 7002.106} C_VEL
LIN {X 0,Y 262.877,Z 965.575,A -85,B 0,C 180,E1 6999.966,E2 6999.966} C_VEL
LIN {X 0,Y 245.402,Z 981.906,A -85,B 0,C 180,E1 6996.974,E2 6996.974} C_VEL
LIN {X 0,Y 228.846,Z 995.882,A -85,B 0,C 180,E1 6993.597,E2 6993.597} C_VEL
LIN {X 0,Y 213.814,Z 1007.712,A -85,B 0,C 180,E1 6989.898,E2 6989.898} C_VEL
LIN {X 0,Y 195.739,Z 1020.888,A -85,B 0,C 180,E1 6984.312,E2 6984.312} C_VEL
LIN {X 0,Y 182.6,Z 1029.892,A -85,B 0,C 180,E1 6979.083,E2 6979.083} C_VEL
LIN {X 0,Y 169.557,Z 1038.647,A -85,B 0,C 180,E1 6972.242,E2 6972.242} C_VEL
LIN {X 0,Y 158.591,Z 1045.886,A -85,B 0,C 180,E1 6964.134,E2 6964.134} C_VEL
LIN {X 0,Y 151.724,Z 1050.715,A -85,B 0,C 180,E1 6956.624,E2 6956.624} C_VEL
LIN {X 0,Y 147.136,Z 1054.428,A -85,B 0,C 180,E1 6948.626,E2 6948.626} C_VEL
LIN {X 0,Y 144.501,Z 1057.394,A -85,B 0,C 180,E1 6939.157,E2 6939.157} C_VEL
LIN {X 0,Y 143.949,Z 1058.738,A -85,B 0,C 180,E1 6930.796,E2 6930.796} C_VEL
LIN {X 0,Y 143.941,Z 1059.074,A -85,B 0,C 180,E1 6923.619,E2 6923.619} C_VEL
LIN {X 0,Y 144.417,Z 1058.49,A -85,B 0,C 180,E1 6915.567,E2 6915.567} C_VEL
LIN {X 0,Y 146.514,Z 1056.812,A -85,B 0,C 180,E1 6907.108,E2 6907.108} C_VEL
LIN {X 0,Y 150.821,Z 1054.04,A -85,B 0,C 180,E1 6898.861,E2 6898.861} C_VEL
LIN {X 0,Y 157.931,Z 1049.941,A -85,B 0,C 180,E1 6890.719,E2 6890.719} C_VEL
LIN {X 0,Y 170.434,Z 1042.919,A -85,B 0,C 180,E1 6881.525,E2 6881.525} C_VEL
LIN {X 0,Y 182.523,Z 1035.983,A -85,B 0,C 180,E1 6875.29,E2 6875.29} C_VEL
LIN {X 0,Y 197.519,Z 1027.072,A -85,B 0,C 180,E1 6869.459,E2 6869.459} C_VEL
LIN {X 0,Y 214.926,Z 1015.825,A -85,B 0,C 180,E1 6864.24,E2 6864.24} C_VEL
LIN {X 0,Y 230.571,Z 1004.942,A -85,B 0,C 180,E1 6860.496,E2 6860.496} C_VEL
LIN {X 0,Y 248.753,Z 991.295,A -85,B 0,C 180,E1 6856.93,E2 6856.93} C_VEL
LIN {X 0,Y 266.87,Z 976.066,A -85,B 0,C 180,E1 6853.976,E2 6853.976} C_VEL
LIN {X 0,Y 281.992,Z 962.223,A -85,B 0,C 180,E1 6851.864,E2 6851.864} C_VEL
LIN {X 0,Y 299.888,Z 944.223,A -85,B 0,C 180,E1 6849.699,E2 6849.699} C_VEL
LIN {X 0,Y 315.815,Z 926.188,A -85,B 0,C 180,E1 6848.008,E2 6848.008} C_VEL
LIN {X 0,Y 329.234,Z 909.462,A -85,B 0,C 180,E1 6846.734,E2 6846.734} C_VEL
LIN {X 0,Y 344.502,Z 888.242,A -85,B 0,C 180,E1 6845.423,E2 6845.423} C_VEL
LIN {X 0,Y 357.027,Z 868.377,A -85,B 0,C 180,E1 6844.433,E2 6844.433} C_VEL
LIN {X 0,Y 367.704,Z 849.41,A -85,B 0,C 180,E1 6843.652,E2 6843.652} C_VEL
LIN {X 0,Y 379.272,Z 826.061,A -85,B 0,C 180,E1 6842.871,E2 6842.871} C_VEL
LIN {X 0,Y 388.757,Z 803.224,A -85,B 0,C 180,E1 6842.257,E2 6842.257} C_VEL
LIN {X 0,Y 396.149,Z 782.401,A -85,B 0,C 180,E1 6841.797,E2 6841.797} C_VEL
LIN {X 0,Y 403.63,Z 756.964,A -85,B 0,C 180,E1 6841.364,E2 6841.364} C_VEL
LIN {X 0,Y 409.143,Z 731.947,A -85,B 0,C 180,E1 6841.024,E2 6841.024} C_VEL
LIN {X 0,Y 412.815,Z 709.422,A -85,B 0,C 180,E1 6840.746,E2 6840.746} C_VEL
LIN {X 0,Y 425.501,Z 605.114,A -85,B 0,C 180,E1 6839.495,E2 6839.495} C_VEL
LIN {X 0,Y 425.477,Z 605.347,A -85,B 0,C 180,E1 6837.553,E2 6837.553} C_VEL
LIN {X 0,Y 411.811,Z 716.574,A -85,B 0,C 180,E1 6836.232,E2 6836.232} C_VEL
LIN {X 0,Y 409.011,Z 732.823,A -85,B 0,C 180,E1 6836.031,E2 6836.031} C_VEL
LIN {X 0,Y 407.519,Z 740.427,A -85,B 0,C 180,E1 6836.091,E2 6836.091} C_VEL
LIN {X 0,Y 402.728,Z 759.514,A -85,B 0,C 180,E1 6836.706,E2 6836.706} C_VEL
LIN {X 0,Y 400.56,Z 766.976,A -85,B 0,C 180,E1 6836.709,E2 6836.709} C_VEL
LIN {X 0,Y 393.506,Z 789.431,A -85,B 0,C 180,E1 6836.343,E2 6836.343} C_VEL
LIN {X 0,Y 383.495,Z 815.412,A -85,B 0,C 180,E1 6835.781,E2 6835.781} C_VEL
LIN {X 0,Y 374.252,Z 835.692,A -85,B 0,C 180,E1 6835.233,E2 6835.233} C_VEL
LIN {X 0,Y 363.594,Z 856.211,A -85,B 0,C 180,E1 6834.564,E2 6834.564} C_VEL
LIN {X 0,Y 349.155,Z 880.269,A -85,B 0,C 180,E1 6833.573,E2 6833.573} C_VEL
LIN {X 0,Y 336.74,Z 898.48,A -85,B 0,C 180,E1 6832.635,E2 6832.635} C_VEL
LIN {X 0,Y 322.538,Z 917.247,A -85,B 0,C 180,E1 6831.462,E2 6831.462} C_VEL
LIN {X 0,Y 305.233,Z 937.503,A -85,B 0,C 180,E1 6829.86,E2 6829.86} C_VEL
LIN {X 0,Y 290.94,Z 952.565,A -85,B 0,C 180,E1 6828.37,E2 6828.37} C_VEL
LIN {X 0,Y 275.527,Z 967.438,A -85,B 0,C 180,E1 6826.549,E2 6826.549} C_VEL
LIN {X 0,Y 255.189,Z 985.119,A -85,B 0,C 180,E1 6823.732,E2 6823.732} C_VEL
LIN {X 0,Y 238.923,Z 997.868,A -85,B 0,C 180,E1 6821.05,E2 6821.05} C_VEL
LIN {X 0,Y 222.448,Z 1009.778,A -85,B 0,C 180,E1 6817.813,E2 6817.813} C_VEL
LIN {X 0,Y 202.986,Z 1022.602,A -85,B 0,C 180,E1 6813.052,E2 6813.052} C_VEL
LIN {X 0,Y 187.921,Z 1031.741,A -85,B 0,C 180,E1 6808.356,E2 6808.356} C_VEL
LIN {X 0,Y 172.996,Z 1040.303,A -85,B 0,C 180,E1 6802.358,E2 6802.358} C_VEL
LIN {X 0,Y 158.658,Z 1048.078,A -85,B 0,C 180,E1 6794.39,E2 6794.39} C_VEL
LIN {X 0,Y 149.049,Z 1053.246,A -85,B 0,C 180,E1 6786.659,E2 6786.659} C_VEL
LIN {X 0,Y 141.812,Z 1057.359,A -85,B 0,C 180,E1 6777.733,E2 6777.733} C_VEL
LIN {X 0,Y 137.237,Z 1060.366,A -85,B 0,C 180,E1 6766.944,E2 6766.944} C_VEL
LIN {X 0,Y 136.012,Z 1061.54,A -85,B 0,C 180,E1 6758.029,E2 6758.029} C_VEL
LIN {X 0,Y 135.918,Z 1061.718,A -85,B 0,C 180,E1 6750.843,E2 6750.843} C_VEL
LIN {X 0,Y 135.928,Z 1061.235,A -85,B 0,C 180,E1 6744.089,E2 6744.089} C_VEL
LIN {X 0,Y 136.66,Z 1059.651,A -85,B 0,C 180,E1 6735.596,E2 6735.596} C_VEL
LIN {X 0,Y 139.363,Z 1056.861,A -85,B 0,C 180,E1 6726.688,E2 6726.688} C_VEL
LIN {X 0,Y 144.421,Z 1052.993,A -85,B 0,C 180,E1 6718.253,E2 6718.253} C_VEL
LIN {X 0,Y 153.278,Z 1047.165,A -85,B 0,C 180,E1 6709.283,E2 6709.283} C_VEL
LIN {X 0,Y 165.637,Z 1039.236,A -85,B 0,C 180,E1 6701.012,E2 6701.012} C_VEL
LIN {X 0,Y 178.145,Z 1031.191,A -85,B 0,C 180,E1 6694.97,E2 6694.97} C_VEL
LIN {X 0,Y 194.414,Z 1020.389,A -85,B 0,C 180,E1 6689.036,E2 6689.036} C_VEL
LIN {X 0,Y 211.574,Z 1007.961,A -85,B 0,C 180,E1 6684.203,E2 6684.203} C_VEL
LIN {X 0,Y 226.696,Z 996.275,A -85,B 0,C 180,E1 6680.762,E2 6680.762} C_VEL
LIN {X 0,Y 245.068,Z 980.854,A -85,B 0,C 180,E1 6677.307,E2 6677.307} C_VEL
LIN {X 0,Y 261.546,Z 965.535,A -85,B 0,C 180,E1 6674.713,E2 6674.713} C_VEL
LIN {X 0,Y 276.695,Z 950.206,A -85,B 0,C 180,E1 6672.66,E2 6672.66} C_VEL
LIN {X 0,Y 294.918,Z 929.686,A -85,B 0,C 180,E1 6670.515,E2 6670.515} C_VEL
LIN {X 0,Y 308.076,Z 913.162,A -85,B 0,C 180,E1 6669.151,E2 6669.151} C_VEL
LIN {X 0,Y 320.51,Z 895.992,A -85,B 0,C 180,E1 6667.976,E2 6667.976} C_VEL
LIN {X 0,Y 335.262,Z 873.159,A -85,B 0,C 180,E1 6666.717,E2 6666.717} C_VEL
LIN {X 0,Y 346.746,Z 852.769,A -85,B 0,C 180,E1 6665.819,E2 6665.819} C_VEL
LIN {X 0,Y 356.383,Z 833.498,A -85,B 0,C 180,E1 6665.126,E2 6665.126} C_VEL
LIN {X 0,Y 366.555,Z 810.226,A -85,B 0,C 180,E1 6664.436,E2 6664.436} C_VEL
LIN {X 0,Y 375.31,Z 785.876,A -85,B 0,C 180,E1 6663.867,E2 6663.867} C_VEL
LIN {X 0,Y 381.846,Z 764.155,A -85,B 0,C 180,E1 6663.479,E2 6663.479} C_VEL
LIN {X 0,Y 388.252,Z 737.072,A -85,B 0,C 180,E1 6663.084,E2 6663.084} C_VEL
LIN {X 0,Y 392.221,Z 713.485,A -85,B 0,C 180,E1 6662.779,E2 6662.779} C_VEL
LIN {X 0,Y 406.185,Z 596.543,A -85,B 0,C 180,E1 6661.34,E2 6661.34} C_VEL
LIN {X 0,Y 405.848,Z 595.026,A -85,B 0,C 180,E1 6658.165,E2 6658.165} C_VEL
LIN {X 0,Y 406.162,Z 596.713,A -85,B 0,C 180,E1 6655.483,E2 6655.483} C_VEL
LIN {X 0,Y 391.841,Z 716.015,A -85,B 0,C 180,E1 6654.036,E2 6654.036} C_VEL
LIN {X 0,Y 386.728,Z 743.945,A -85,B 0,C 180,E1 6653.668,E2 6653.668} C_VEL
LIN {X 0,Y 381.022,Z 766.706,A -85,B 0,C 180,E1 6653.305,E2 6653.305} C_VEL
LIN {X 0,Y 374.587,Z 787.687,A -85,B 0,C 180,E1 6652.89,E2 6652.89} C_VEL
LIN {X 0,Y 364.804,Z 813.907,A -85,B 0,C 180,E1 6652.233,E2 6652.233} C_VEL
LIN {X 0,Y 355.784,Z 834.241,A -85,B 0,C 180,E1 6651.591,E2 6651.591} C_VEL
LIN {X 0,Y 346.122,Z 853.411,A -85,B 0,C 180,E1 6650.858,E2 6650.858} C_VEL
LIN {X 0,Y 332.997,Z 876.305,A -85,B 0,C 180,E1 6649.796,E2 6649.796} C_VEL
LIN {X 0,Y 319.851,Z 896.249,A -85,B 0,C 180,E1 6648.642,E2 6648.642} C_VEL
LIN {X 0,Y 307.003,Z 913.831,A -85,B 0,C 180,E1 6647.396,E2 6647.396} C_VEL
LIN {X 0,Y 290.569,Z 934.031,A -85,B 0,C 180,E1 6645.621,E2 6645.621} C_VEL
LIN {X 0,Y 275,Z 951.042,A -85,B 0,C 180,E1 6643.717,E2 6643.717} C_VEL
LIN {X 0,Y 259.947,Z 966.087,A -85,B 0,C 180,E1 6641.614,E2 6641.614} C_VEL
LIN {X 0,Y 240.764,Z 983.44,A -85,B 0,C 180,E1 6638.476,E2 6638.476} C_VEL
LIN {X 0,Y 225.328,Z 996.103,A -85,B 0,C 180,E1 6635.461,E2 6635.461} C_VEL
LIN {X 0,Y 209.824,Z 1007.92,A -85,B 0,C 180,E1 6631.835,E2 6631.835} C_VEL
LIN {X 0,Y 191.756,Z 1020.618,A -85,B 0,C 180,E1 6626.542,E2 6626.542} C_VEL
LIN {X 0,Y 177.958,Z 1029.665,A -85,B 0,C 180,E1 6621.351,E2 6621.351} C_VEL
LIN {X 0,Y 165.17,Z 1037.763,A -85,B 0,C 180,E1 6615.095,E2 6615.095} C_VEL
LIN {X 0,Y 152.305,Z 1045.773,A -85,B 0,C 180,E1 6606.217,E2 6606.217} C_VEL
LIN {X 0,Y 144.493,Z 1050.841,A -85,B 0,C 180,E1 6598.07,E2 6598.07} C_VEL
LIN {X 0,Y 139.304,Z 1054.7,A -85,B 0,C 180,E1 6589.279,E2 6589.279} C_VEL
LIN {X 0,Y 136.505,Z 1057.582,A -85,B 0,C 180,E1 6579.273,E2 6579.273} C_VEL
LIN {X 0,Y 135.948,Z 1058.821,A -85,B 0,C 180,E1 6570.843,E2 6570.843} C_VEL
LIN {X 0,Y 135.94,Z 1059.169,A -85,B 0,C 180,E1 6563.665,E2 6563.665} C_VEL
LIN {X 0,Y 136.464,Z 1058.621,A -85,B 0,C 180,E1 6555.14,E2 6555.14} C_VEL
LIN {X 0,Y 138.946,Z 1056.866,A -85,B 0,C 180,E1 6545.783,E2 6545.783} C_VEL
LIN {X 0,Y 143.746,Z 1054.084,A -85,B 0,C 180,E1 6537.142,E2 6537.142} C_VEL
LIN {X 0,Y 151.532,Z 1049.975,A -85,B 0,C 180,E1 6528.711,E2 6528.711} C_VEL
LIN {X 0,Y 164.627,Z 1043.116,A -85,B 0,C 180,E1 6519.524,E2 6519.524} C_VEL
LIN {X 0,Y 177.781,Z 1035.983,A -85,B 0,C 180,E1 6513.069,E2 6513.069} C_VEL
LIN {X 0,Y 193.506,Z 1027.061,A -85,B 0,C 180,E1 6507.282,E2 6507.282} C_VEL
LIN {X 0,Y 211.601,Z 1015.789,A -85,B 0,C 180,E1 6502.156,E2 6502.156} C_VEL
LIN {X 0,Y 226.93,Z 1005.468,A -85,B 0,C 180,E1 6498.681,E2 6498.681} C_VEL
LIN {X 0,Y 244.706,Z 992.522,A -85,B 0,C 180,E1 6495.353,E2 6495.353} C_VEL
LIN {X 0,Y 263.182,Z 977.521,A -85,B 0,C 180,E1 6492.473,E2 6492.473} C_VEL
LIN {X 0,Y 278.564,Z 963.813,A -85,B 0,C 180,E1 6490.421,E2 6490.421} C_VEL
LIN {X 0,Y 294.735,Z 948.06,A -85,B 0,C 180,E1 6488.541,E2 6488.541} C_VEL
LIN {X 0,Y 312.697,Z 928.461,A -85,B 0,C 180,E1 6486.712,E2 6486.712} C_VEL
LIN {X 0,Y 326.448,Z 911.724,A -85,B 0,C 180,E1 6485.468,E2 6485.468} C_VEL
LIN {X 0,Y 339.942,Z 893.572,A -85,B 0,C 180,E1 6484.354,E2 6484.354} C_VEL
LIN {X 0,Y 354.928,Z 870.71,A -85,B 0,C 180,E1 6483.23,E2 6483.23} C_VEL
LIN {X 0,Y 366.291,Z 850.911,A -85,B 0,C 180,E1 6482.444,E2 6482.444} C_VEL
LIN {X 0,Y 376.762,Z 830.27,A -85,B 0,C 180,E1 6481.774,E2 6481.774} C_VEL
LIN {X 0,Y 387.529,Z 805.334,A -85,B 0,C 180,E1 6481.117,E2 6481.117} C_VEL
LIN {X 0,Y 395.231,Z 784.076,A -85,B 0,C 180,E1 6480.665,E2 6480.665} C_VEL
LIN {X 0,Y 402.056,Z 761.575,A -85,B 0,C 180,E1 6480.293,E2 6480.293} C_VEL
LIN {X 0,Y 408.422,Z 734.343,A -85,B 0,C 180,E1 6479.929,E2 6479.929} C_VEL
LIN {X 0,Y 412.225,Z 711.916,A -85,B 0,C 180,E1 6479.662,E2 6479.662} C_VEL
LIN {X 0,Y 424.301,Z 614.4,A -85,B 0,C 180,E1 6478.532,E2 6478.532} C_VEL
LIN {X 0,Y 411.542,Z 716.705,A -85,B 0,C 180,E1 6477.347,E2 6477.347} C_VEL
LIN {X 0,Y 406.103,Z 745.372,A -85,B 0,C 180,E1 6477,E2 6477} C_VEL
LIN {X 0,Y 400.56,Z 766.976,A -85,B 0,C 180,E1 6476.709,E2 6476.709} C_VEL
LIN {X 0,Y 398.739,Z 773.359,A -85,B 0,C 180,E1 6476.739,E2 6476.739} C_VEL
LIN {X 0,Y 391.59,Z 794.301,A -85,B 0,C 180,E1 6477.315,E2 6477.315} C_VEL
LIN {X 0,Y 389.236,Z 800.348,A -85,B 0,C 180,E1 6477.307,E2 6477.307} C_VEL
LIN {X 0,Y 380.532,Z 821.423,A -85,B 0,C 180,E1 6476.847,E2 6476.847} C_VEL
LIN {X 0,Y 368.779,Z 845.777,A -85,B 0,C 180,E1 6476.175,E2 6476.175} C_VEL
LIN {X 0,Y 357.079,Z 866.512,A -85,B 0,C 180,E1 6475.461,E2 6475.461} C_VEL
LIN {X 0,Y 345.22,Z 885.214,A -85,B 0,C 180,E1 6474.682,E2 6474.682} C_VEL
LIN {X 0,Y 329.803,Z 906.833,A -85,B 0,C 180,E1 6473.559,E2 6473.559} C_VEL
LIN {X 0,Y 314.594,Z 925.556,A -85,B 0,C 180,E1 6472.329,E2 6472.329} C_VEL
LIN {X 0,Y 300.142,Z 941.674,A -85,B 0,C 180,E1 6471.022,E2 6471.022} C_VEL
LIN {X 0,Y 282,Z 959.965,A -85,B 0,C 180,E1 6469.16,E2 6469.16} C_VEL
LIN {X 0,Y 264.649,Z 975.509,A -85,B 0,C 180,E1 6467.101,E2 6467.101} C_VEL
LIN {X 0,Y 248.575,Z 988.677,A -85,B 0,C 180,E1 6464.882,E2 6464.882} C_VEL
LIN {X 0,Y 229.258,Z 1003.138,A -85,B 0,C 180,E1 6461.698,E2 6461.698} C_VEL
LIN {X 0,Y 210.458,Z 1015.681,A -85,B 0,C 180,E1 6457.887,E2 6457.887} C_VEL
LIN {X 0,Y 194.777,Z 1025.354,A -85,B 0,C 180,E1 6453.943,E2 6453.943} C_VEL
LIN {X 0,Y 176.659,Z 1035.701,A -85,B 0,C 180,E1 6448.103,E2 6448.103} C_VEL
LIN {X 0,Y 161.853,Z 1043.465,A -85,B 0,C 180,E1 6441.681,E2 6441.681} C_VEL
LIN {X 0,Y 149.759,Z 1049.583,A -85,B 0,C 180,E1 6434.511,E2 6434.511} C_VEL
LIN {X 0,Y 138.648,Z 1055.224,A -85,B 0,C 180,E1 6424.7,E2 6424.7} C_VEL
LIN {X 0,Y 131.847,Z 1058.79,A -85,B 0,C 180,E1 6414.488,E2 6414.488} C_VEL
LIN {X 0,Y 128.923,Z 1060.649,A -85,B 0,C 180,E1 6405.751,E2 6405.751} C_VEL
LIN {X 0,Y 127.99,Z 1061.514,A -85,B 0,C 180,E1 6397.632,E2 6397.632} C_VEL
LIN {X 0,Y 127.917,Z 1061.635,A -85,B 0,C 180,E1 6390.896,E2 6390.896} C_VEL
LIN {X 0,Y 127.937,Z 1061.143,A -85,B 0,C 180,E1 6383.719,E2 6383.719} C_VEL
LIN {X 0,Y 128.802,Z 1059.548,A -85,B 0,C 180,E1 6374.696,E2 6374.696} C_VEL
LIN {X 0,Y 131.828,Z 1056.773,A -85,B 0,C 180,E1 6365.345,E2 6365.345} C_VEL
LIN {X 0,Y 137.462,Z 1052.869,A -85,B 0,C 180,E1 6356.44,E2 6356.44} C_VEL
LIN {X 0,Y 147.542,Z 1046.771,A -85,B 0,C 180,E1 6346.806,E2 6346.806} C_VEL
LIN {X 0,Y 160.971,Z 1038.662,A -85,B 0,C 180,E1 6338.401,E2 6338.401} C_VEL
LIN {X 0,Y 174.162,Z 1030.612,A -85,B 0,C 180,E1 6332.441,E2 6332.441} C_VEL
LIN {X 0,Y 191.99,Z 1019.154,A -85,B 0,C 180,E1 6326.392,E2 6326.392} C_VEL
LIN {X 0,Y 208.285,Z 1007.757,A -85,B 0,C 180,E1 6322.104,E2 6322.104} C_VEL
LIN {X 0,Y 224.711,Z 995.414,A -85,B 0,C 180,E1 6318.6,E2 6318.6} C_VEL
LIN {X 0,Y 244.469,Z 979.048,A -85,B 0,C 180,E1 6315.151,E2 6315.151} C_VEL
LIN {X 0,Y 259.88,Z 964.969,A -85,B 0,C 180,E1 6312.895,E2 6312.895} C_VEL
LIN {X 0,Y 275.966,Z 948.939,A -85,B 0,C 180,E1 6310.86,E2 6310.86} C_VEL
LIN {X 0,Y 293.785,Z 929.055,A -85,B 0,C 180,E1 6308.902,E2 6308.902} C_VEL
LIN {X 0,Y 307.166,Z 912.441,A -85,B 0,C 180,E1 6307.605,E2 6307.605} C_VEL
LIN {X 0,Y 320.273,Z 894.5,A -85,B 0,C 180,E1 6306.453,E2 6306.453} C_VEL
LIN {X 0,Y 335.368,Z 871.091,A -85,B 0,C 180,E1 6305.251,E2 6305.251} C_VEL
LIN {X 0,Y 346.499,Z 851.395,A -85,B 0,C 180,E1 6304.439,E2 6304.439} C_VEL
LIN {X 0,Y 357.7,Z 828.929,A -85,B 0,C 180,E1 6303.692,E2 6303.692} C_VEL
LIN {X 0,Y 367.938,Z 804.516,A -85,B 0,C 180,E1 6303.05,E2 6303.05} C_VEL
LIN {X 0,Y 375.097,Z 784.42,A -85,B 0,C 180,E1 6302.617,E2 6302.617} C_VEL
LIN {X 0,Y 382.167,Z 760.758,A -85,B 0,C 180,E1 6302.223,E2 6302.223} C_VEL
LIN {X 0,Y 388.253,Z 734,A -85,B 0,C 180,E1 6301.864,E2 6301.864} C_VEL
LIN {X 0,Y 391.935,Z 711.767,A -85,B 0,C 180,E1 6301.588,E2 6301.588} C_VEL
LIN {X 0,Y 404.967,Z 603.911,A -85,B 0,C 180,E1 6300.283,E2 6300.283} C_VEL
LIN {X 0,Y 404.87,Z 602.987,A -85,B 0,C 180,E1 6298.16,E2 6298.16} C_VEL
LIN {X 0,Y 404.945,Z 604.103,A -85,B 0,C 180,E1 6296.529,E2 6296.529} C_VEL
LIN {X 0,Y 391.284,Z 716.231,A -85,B 0,C 180,E1 6295.204,E2 6295.204} C_VEL
LIN {X 0,Y 386.054,Z 744.389,A -85,B 0,C 180,E1 6294.849,E2 6294.849} C_VEL
LIN {X 0,Y 380.358,Z 766.878,A -85,B 0,C 180,E1 6294.507,E2 6294.507} C_VEL
LIN {X 0,Y 373.925,Z 787.663,A -85,B 0,C 180,E1 6294.118,E2 6294.118} C_VEL
LIN {X 0,Y 363.81,Z 814.468,A -85,B 0,C 180,E1 6293.48,E2 6293.48} C_VEL
LIN {X 0,Y 354.702,Z 834.749,A -85,B 0,C 180,E1 6292.869,E2 6292.869} C_VEL
LIN {X 0,Y 344.542,Z 854.62,A -85,B 0,C 180,E1 6292.144,E2 6292.144} C_VEL
LIN {X 0,Y 330.468,Z 878.545,A -85,B 0,C 180,E1 6291.069,E2 6291.069} C_VEL
LIN {X 0,Y 317.778,Z 897.441,A -85,B 0,C 180,E1 6290.014,E2 6290.014} C_VEL
LIN {X 0,Y 303.824,Z 916.151,A -85,B 0,C 180,E1 6288.73,E2 6288.73} C_VEL
LIN {X 0,Y 286.837,Z 936.339,A -85,B 0,C 180,E1 6286.984,E2 6286.984} C_VEL
LIN {X 0,Y 271.937,Z 952.241,A -85,B 0,C 180,E1 6285.245,E2 6285.245} C_VEL
LIN {X 0,Y 255.999,Z 967.78,A -85,B 0,C 180,E1 6283.122,E2 6283.122} C_VEL
LIN {X 0,Y 237.04,Z 984.368,A -85,B 0,C 180,E1 6280.162,E2 6280.162} C_VEL
LIN {X 0,Y 221.238,Z 996.951,A -85,B 0,C 180,E1 6277.217,E2 6277.217} C_VEL
LIN {X 0,Y 203.76,Z 1009.826,A -85,B 0,C 180,E1 6273.266,E2 6273.266} C_VEL
LIN {X 0,Y 185.929,Z 1021.705,A -85,B 0,C 180,E1 6268.178,E2 6268.178} C_VEL
LIN {X 0,Y 171.656,Z 1030.634,A -85,B 0,C 180,E1 6262.941,E2 6262.941} C_VEL
LIN {X 0,Y 156.707,Z 1039.605,A -85,B 0,C 180,E1 6255.612,E2 6255.612} C_VEL
LIN {X 0,Y 144.916,Z 1046.41,A -85,B 0,C 180,E1 6247.385,E2 6247.385} C_VEL
LIN {X 0,Y 136.728,Z 1051.373,A -85,B 0,C 180,E1 6238.859,E2 6238.859} C_VEL
LIN {X 0,Y 130.789,Z 1055.589,A -85,B 0,C 180,E1 6228.267,E2 6228.267} C_VEL
LIN {X 0,Y 128.336,Z 1057.941,A -85,B 0,C 180,E1 6218.062,E2 6218.062} C_VEL
LIN {X 0,Y 127.943,Z 1058.948,A -85,B 0,C 180,E1 6210,E2 6210} C_VEL
LIN {X 0,Y 127.957,Z 1059.22,A -85,B 0,C 180,E1 6202.817,E2 6202.817} C_VEL
LIN {X 0,Y 128.658,Z 1058.618,A -85,B 0,C 180,E1 6193.753,E2 6193.753} C_VEL
LIN {X 0,Y 131.437,Z 1056.92,A -85,B 0,C 180,E1 6184.302,E2 6184.302} C_VEL
LIN {X 0,Y 136.812,Z 1054.128,A -85,B 0,C 180,E1 6175.245,E2 6175.245} C_VEL
LIN {X 0,Y 145.782,Z 1049.803,A -85,B 0,C 180,E1 6166.153,E2 6166.153} C_VEL
LIN {X 0,Y 159.391,Z 1043.128,A -85,B 0,C 180,E1 6157.184,E2 6157.184} C_VEL
LIN {X 0,Y 172.646,Z 1036.338,A -85,B 0,C 180,E1 6151.002,E2 6151.002} C_VEL
LIN {X 0,Y 188.285,Z 1027.862,A -85,B 0,C 180,E1 6145.474,E2 6145.474} C_VEL
LIN {X 0,Y 207.756,Z 1016.269,A -85,B 0,C 180,E1 6140.2,E2 6140.2} C_VEL
LIN {X 0,Y 224.376,Z 1005.419,A -85,B 0,C 180,E1 6136.644,E2 6136.644} C_VEL
LIN {X 0,Y 243.6,Z 991.753,A -85,B 0,C 180,E1 6133.289,E2 6133.289} C_VEL
LIN {X 0,Y 262.416,Z 976.652,A -85,B 0,C 180,E1 6130.562,E2 6130.562} C_VEL
LIN {X 0,Y 278.107,Z 962.853,A -85,B 0,C 180,E1 6128.617,E2 6128.617} C_VEL
LIN {X 0,Y 296.461,Z 945.089,A -85,B 0,C 180,E1 6126.65,E2 6126.65} C_VEL
LIN {X 0,Y 313.193,Z 926.72,A -85,B 0,C 180,E1 6125.078,E2 6125.078} C_VEL
LIN {X 0,Y 327.221,Z 909.698,A -85,B 0,C 180,E1 6123.903,E2 6123.903} C_VEL
LIN {X 0,Y 342.848,Z 888.496,A -85,B 0,C 180,E1 6122.725,E2 6122.725} C_VEL
LIN {X 0,Y 355.642,Z 868.643,A -85,B 0,C 180,E1 6121.836,E2 6121.836} C_VEL
LIN {X 0,Y 366.529,Z 849.689,A -85,B 0,C 180,E1 6121.133,E2 6121.133} C_VEL
LIN {X 0,Y 377.988,Z 827.077,A -85,B 0,C 180,E1 6120.455,E2 6120.455} C_VEL
LIN {X 0,Y 387.956,Z 803.559,A -85,B 0,C 180,E1 6119.888,E2 6119.888} C_VEL
LIN {X 0,Y 395.471,Z 782.765,A -85,B 0,C 180,E1 6119.474,E2 6119.474} C_VEL
LIN {X 0,Y 403.036,Z 757.546,A -85,B 0,C 180,E1 6119.09,E2 6119.09} C_VEL
LIN {X 0,Y 408.733,Z 732.143,A -85,B 0,C 180,E1 6118.778,E2 6118.778} C_VEL
LIN {X 0,Y 412.276,Z 711.036,A -85,B 0,C 180,E1 6118.529,E2 6118.529} C_VEL
LIN {X 0,Y 408.513,Z 733.306,A -85,B 0,C 180,E1 6118.274,E2 6118.274} C_VEL
LIN {X 0,Y 402.49,Z 759.579,A -85,B 0,C 180,E1 6117.96,E2 6117.96} C_VEL
LIN {X 0,Y 395.297,Z 783.361,A -85,B 0,C 180,E1 6117.613,E2 6117.613} C_VEL
LIN {X 0,Y 389.236,Z 800.348,A -85,B 0,C 180,E1 6117.307,E2 6117.307} C_VEL
LIN {X 0,Y 386.373,Z 807.742,A -85,B 0,C 180,E1 6117.305,E2 6117.305} C_VEL
LIN {X 0,Y 378.439,Z 825.798,A -85,B 0,C 180,E1 6117.81,E2 6117.81} C_VEL
LIN {X 0,Y 375.067,Z 832.727,A -85,B 0,C 180,E1 6117.788,E2 6117.788} C_VEL
LIN {X 0,Y 364.963,Z 852.195,A -85,B 0,C 180,E1 6117.243,E2 6117.243} C_VEL
LIN {X 0,Y 353.101,Z 872.421,A -85,B 0,C 180,E1 6116.545,E2 6116.545} C_VEL
LIN {X 0,Y 337.965,Z 894.908,A -85,B 0,C 180,E1 6115.583,E2 6115.583} C_VEL
LIN {X 0,Y 324.384,Z 912.77,A -85,B 0,C 180,E1 6114.634,E2 6114.634} C_VEL
LIN {X 0,Y 308.993,Z 931.028,A -85,B 0,C 180,E1 6113.431,E2 6113.431} C_VEL
LIN {X 0,Y 290.917,Z 950.039,A -85,B 0,C 180,E1 6111.834,E2 6111.834} C_VEL
LIN {X 0,Y 274.966,Z 965.115,A -85,B 0,C 180,E1 6110.218,E2 6110.218} C_VEL
LIN {X 0,Y 258.35,Z 979.431,A -85,B 0,C 180,E1 6108.287,E2 6108.287} C_VEL
LIN {X 0,Y 237.615,Z 995.445,A -85,B 0,C 180,E1 6105.43,E2 6105.43} C_VEL
LIN {X 0,Y 220.552,Z 1007.304,A -85,B 0,C 180,E1 6102.589,E2 6102.589} C_VEL
LIN {X 0,Y 202.523,Z 1018.793,A -85,B 0,C 180,E1 6098.927,E2 6098.927} C_VEL
LIN {X 0,Y 182.753,Z 1030.132,A -85,B 0,C 180,E1 6093.803,E2 6093.803} C_VEL
LIN {X 0,Y 167.462,Z 1038.171,A -85,B 0,C 180,E1 6088.63,E2 6088.63} C_VEL
LIN {X 0,Y 151.887,Z 1045.879,A -85,B 0,C 180,E1 6081.572,E2 6081.572} C_VEL
LIN {X 0,Y 137.775,Z 1052.414,A -85,B 0,C 180,E1 6072.247,E2 6072.247} C_VEL
LIN {X 0,Y 129.061,Z 1056.458,A -85,B 0,C 180,E1 6063.372,E2 6063.372} C_VEL
LIN {X 0,Y 123.226,Z 1059.386,A -85,B 0,C 180,E1 6053.428,E2 6053.428} C_VEL
LIN {X 0,Y 120.298,Z 1061.247,A -85,B 0,C 180,E1 6041.993,E2 6041.993} C_VEL
LIN {X 0,Y 119.906,Z 1061.662,A -85,B 0,C 180,E1 6033.347,E2 6033.347} C_VEL
LIN {X 0,Y 119.907,Z 1061.348,A -85,B 0,C 180,E1 6026.654,E2 6026.654} C_VEL
LIN {X 0,Y 120.234,Z 1060.358,A -85,B 0,C 180,E1 6018.487,E2 6018.487} C_VEL
LIN {X 0,Y 122.783,Z 1057.938,A -85,B 0,C 180,E1 6007.497,E2 6007.497} C_VEL
LIN {X 0,Y 129.24,Z 1053.587,A -85,B 0,C 180,E1 5996.149,E2 5996.149} C_VEL
LIN {X 0,Y 137.695,Z 1048.708,A -85,B 0,C 180,E1 5987.521,E2 5987.521} C_VEL
LIN {X 0,Y 150.356,Z 1041.714,A -85,B 0,C 180,E1 5978.917,E2 5978.917} C_VEL
LIN {X 0,Y 166.341,Z 1032.499,A -85,B 0,C 180,E1 5971.398,E2 5971.398} C_VEL
LIN {X 0,Y 181.331,Z 1023.421,A -85,B 0,C 180,E1 5966.176,E2 5966.176} C_VEL
LIN {X 0,Y 199.562,Z 1011.621,A -85,B 0,C 180,E1 5961.262,E2 5961.262} C_VEL
LIN {X 0,Y 217.964,Z 998.367,A -85,B 0,C 180,E1 5957.349,E2 5957.349} C_VEL
LIN {X 0,Y 233.54,Z 986.212,A -85,B 0,C 180,E1 5954.625,E2 5954.625} C_VEL
LIN {X 0,Y 252.36,Z 970.146,A -85,B 0,C 180,E1 5951.862,E2 5951.862} C_VEL
LIN {X 0,Y 269.821,Z 953.398,A -85,B 0,C 180,E1 5949.693,E2 5949.693} C_VEL
LIN {X 0,Y 284.322,Z 938.148,A -85,B 0,C 180,E1 5948.127,E2 5948.127} C_VEL
LIN {X 0,Y 300.925,Z 918.867,A -85,B 0,C 180,E1 5946.543,E2 5946.543} C_VEL
LIN {X 0,Y 315.902,Z 899.093,A -85,B 0,C 180,E1 5945.267,E2 5945.267} C_VEL
LIN {X 0,Y 328.389,Z 880.776,A -85,B 0,C 180,E1 5944.308,E2 5944.308} C_VEL
LIN {X 0,Y 342.535,Z 857.295,A -85,B 0,C 180,E1 5943.321,E2 5943.321} C_VEL
LIN {X 0,Y 353.33,Z 836.539,A -85,B 0,C 180,E1 5942.629,E2 5942.629} C_VEL
LIN {X 0,Y 362.509,Z 816.422,A -85,B 0,C 180,E1 5942.071,E2 5942.071} C_VEL
LIN {X 0,Y 372.336,Z 791.178,A -85,B 0,C 180,E1 5941.515,E2 5941.515} C_VEL
LIN {X 0,Y 379.722,Z 767.752,A -85,B 0,C 180,E1 5941.126,E2 5941.126} C_VEL
LIN {X 0,Y 385.307,Z 746.022,A -85,B 0,C 180,E1 5940.829,E2 5940.829} C_VEL
LIN {X 0,Y 390.702,Z 717.848,A -85,B 0,C 180,E1 5940.487,E2 5940.487} C_VEL
LIN {X 0,Y 399.691,Z 645.888,A -85,B 0,C 180,E1 5939.657,E2 5939.657} C_VEL
LIN {X 0,Y 403.892,Z 611.271,A -85,B 0,C 180,E1 5939.255,E2 5939.255} C_VEL
LIN {X 0,Y 403.892,Z 610.951,A -85,B 0,C 180,E1 5938.156,E2 5938.156} C_VEL
LIN {X 0,Y 403.871,Z 611.426,A -85,B 0,C 180,E1 5937.581,E2 5937.581} C_VEL
LIN {X 0,Y 390.892,Z 716.435,A -85,B 0,C 180,E1 5936.376,E2 5936.376} C_VEL
LIN {X 0,Y 385.511,Z 744.977,A -85,B 0,C 180,E1 5936.031,E2 5936.031} C_VEL
LIN {X 0,Y 379.801,Z 767.265,A -85,B 0,C 180,E1 5935.71,E2 5935.71} C_VEL
LIN {X 0,Y 373.192,Z 788.372,A -85,B 0,C 180,E1 5935.335,E2 5935.335} C_VEL
LIN {X 0,Y 362.99,Z 815.03,A -85,B 0,C 180,E1 5934.733,E2 5934.733} C_VEL
LIN {X 0,Y 353.798,Z 835.257,A -85,B 0,C 180,E1 5934.155,E2 5934.155} C_VEL
LIN {X 0,Y 343.802,Z 854.594,A -85,B 0,C 180,E1 5933.487,E2 5933.487} C_VEL
LIN {X 0,Y 329.315,Z 878.94,A -85,B 0,C 180,E1 5932.452,E2 5932.452} C_VEL
LIN {X 0,Y 316.479,Z 897.808,A -85,B 0,C 180,E1 5931.452,E2 5931.452} C_VEL
LIN {X 0,Y 302.349,Z 916.492,A -85,B 0,C 180,E1 5930.231,E2 5930.231} C_VEL
LIN {X 0,Y 285.31,Z 936.435,A -85,B 0,C 180,E1 5928.59,E2 5928.59} C_VEL
LIN {X 0,Y 270.456,Z 952.049,A -85,B 0,C 180,E1 5926.966,E2 5926.966} C_VEL
LIN {X 0,Y 254.35,Z 967.488,A -85,B 0,C 180,E1 5924.962,E2 5924.962} C_VEL
LIN {X 0,Y 235.263,Z 983.911,A -85,B 0,C 180,E1 5922.178,E2 5922.178} C_VEL
LIN {X 0,Y 219.04,Z 996.545,A -85,B 0,C 180,E1 5919.356,E2 5919.356} C_VEL
LIN {X 0,Y 202.606,Z 1008.335,A -85,B 0,C 180,E1 5915.922,E2 5915.922} C_VEL
LIN {X 0,Y 183.22,Z 1020.983,A -85,B 0,C 180,E1 5910.828,E2 5910.828} C_VEL
LIN {X 0,Y 168.199,Z 1030.005,A -85,B 0,C 180,E1 5905.721,E2 5905.721} C_VEL
LIN {X 0,Y 153.438,Z 1038.429,A -85,B 0,C 180,E1 5899.105,E2 5899.105} C_VEL
LIN {X 0,Y 139.449,Z 1046.047,A -85,B 0,C 180,E1 5890.19,E2 5890.19} C_VEL
LIN {X 0,Y 130.344,Z 1051.092,A -85,B 0,C 180,E1 5881.442,E2 5881.442} C_VEL
LIN {X 0,Y 123.911,Z 1055.087,A -85,B 0,C 180,E1 5871.292,E2 5871.292} C_VEL
LIN {X 0,Y 120.584,Z 1057.835,A -85,B 0,C 180,E1 5860.028,E2 5860.028} C_VEL
LIN {X 0,Y 119.953,Z 1059.008,A -85,B 0,C 180,E1 5850.477,E2 5850.477} C_VEL
LIN {X 0,Y 119.957,Z 1059.311,A -85,B 0,C 180,E1 5842.712,E2 5842.712} C_VEL
LIN {X 0,Y 120.737,Z 1058.749,A -85,B 0,C 180,E1 5833.151,E2 5833.151} C_VEL
LIN {X 0,Y 124.021,Z 1056.975,A -85,B 0,C 180,E1 5822.642,E2 5822.642} C_VEL
LIN {X 0,Y 130.118,Z 1054.138,A -85,B 0,C 180,E1 5813.053,E2 5813.053} C_VEL
LIN {X 0,Y 140.846,Z 1049.426,A -85,B 0,C 180,E1 5803.012,E2 5803.012} C_VEL
LIN {X 0,Y 155.064,Z 1042.838,A -85,B 0,C 180,E1 5794.374,E2 5794.374} C_VEL
LIN {X 0,Y 169.446,Z 1035.846,A -85,B 0,C 180,E1 5788.169,E2 5788.169} C_VEL
LIN {X 0,Y 187.935,Z 1026.188,A -85,B 0,C 180,E1 5782.219,E2 5782.219} C_VEL
LIN {X 0,Y 206.676,Z 1015.2,A -85,B 0,C 180,E1 5777.622,E2 5777.622} C_VEL
LIN {X 0,Y 222.989,Z 1004.794,A -85,B 0,C 180,E1 5774.409,E2 5774.409} C_VEL
LIN {X 0,Y 243.292,Z 990.543,A -85,B 0,C 180,E1 5771.137,E2 5771.137} C_VEL
LIN {X 0,Y 261.014,Z 976.56,A -85,B 0,C 180,E1 5768.758,E2 5768.758} C_VEL
LIN {X 0,Y 276.982,Z 962.745,A -85,B 0,C 180,E1 5766.912,E2 5766.912} C_VEL
LIN {X 0,Y 295.69,Z 944.864,A -85,B 0,C 180,E1 5765.044,E2 5765.044} C_VEL
LIN {X 0,Y 312.569,Z 926.555,A -85,B 0,C 180,E1 5763.565,E2 5763.565} C_VEL
LIN {X 0,Y 326.808,Z 909.454,A -85,B 0,C 180,E1 5762.455,E2 5762.455} C_VEL
LIN {X 0,Y 343.051,Z 887.512,A -85,B 0,C 180,E1 5761.316,E2 5761.316} C_VEL
LIN {X 0,Y 355.473,Z 868.367,A -85,B 0,C 180,E1 5760.516,E2 5760.516} C_VEL
LIN {X 0,Y 366.659,Z 849.011,A -85,B 0,C 180,E1 5759.844,E2 5759.844} C_VEL
LIN {X 0,Y 378.681,Z 825.168,A -85,B 0,C 180,E1 5759.18,E2 5759.18} C_VEL
LIN {X 0,Y 388.057,Z 803.079,A -85,B 0,C 180,E1 5758.687,E2 5758.687} C_VEL
LIN {X 0,Y 390.501,Z 796.803,A -85,B 0,C 180,E1 5758.564,E2 5758.564} C_VEL
LIN {X 0,Y 381.66,Z 818.453,A -85,B 0,C 180,E1 5758.126,E2 5758.126} C_VEL
LIN {X 0,Y 375.067,Z 832.727,A -85,B 0,C 180,E1 5757.788,E2 5757.788} C_VEL
LIN {X 0,Y 371.578,Z 839.771,A -85,B 0,C 180,E1 5757.758,E2 5757.758} C_VEL
LIN {X 0,Y 362.085,Z 857.194,A -85,B 0,C 180,E1 5758.21,E2 5758.21} C_VEL
LIN {X 0,Y 358.135,Z 863.83,A -85,B 0,C 180,E1 5758.158,E2 5758.158} C_VEL
LIN {X 0,Y 345.799,Z 883.159,A -85,B 0,C 180,E1 5757.465,E2 5757.465} C_VEL
LIN {X 0,Y 332.532,Z 901.75,A -85,B 0,C 180,E1 5756.644,E2 5756.644} C_VEL
LIN {X 0,Y 314.96,Z 923.458,A -85,B 0,C 180,E1 5755.442,E2 5755.442} C_VEL
LIN {X 0,Y 299.906,Z 939.982,A -85,B 0,C 180,E1 5754.285,E2 5754.285} C_VEL
LIN {X 0,Y 283.18,Z 956.608,A -85,B 0,C 180,E1 5752.833,E2 5752.833} C_VEL
LIN {X 0,Y 263.226,Z 974.235,A -85,B 0,C 180,E1 5750.82,E2 5750.82} C_VEL
LIN {X 0,Y 246.623,Z 987.421,A -85,B 0,C 180,E1 5748.855,E2 5748.855} C_VEL
LIN {X 0,Y 228.456,Z 1000.564,A -85,B 0,C 180,E1 5746.32,E2 5746.32} C_VEL
LIN {X 0,Y 207.353,Z 1014.198,A -85,B 0,C 180,E1 5742.705,E2 5742.705} C_VEL
LIN {X 0,Y 189.694,Z 1024.471,A -85,B 0,C 180,E1 5738.903,E2 5738.903} C_VEL
LIN {X 0,Y 170.727,Z 1034.594,A -85,B 0,C 180,E1 5733.645,E2 5733.645} C_VEL
LIN {X 0,Y 152.759,Z 1043.128,A -85,B 0,C 180,E1 5726.912,E2 5726.912} C_VEL
LIN {X 0,Y 139.556,Z 1049.019,A -85,B 0,C 180,E1 5720.053,E2 5720.053} C_VEL
LIN {X 0,Y 126.724,Z 1054.591,A -85,B 0,C 180,E1 5710.316,E2 5710.316} C_VEL
LIN {X 0,Y 117.454,Z 1058.522,A -85,B 0,C 180,E1 5698.472,E2 5698.472} C_VEL
LIN {X 0,Y 113.469,Z 1060.449,A -85,B 0,C 180,E1 5688.496,E2 5688.496} C_VEL
LIN {X 0,Y 112.072,Z 1061.342,A -85,B 0,C 180,E1 5679.241,E2 5679.241} C_VEL
LIN {X 0,Y 111.91,Z 1061.493,A -85,B 0,C 180,E1 5671.536,E2 5671.536} C_VEL
LIN {X 0,Y 111.932,Z 1061.097,A -85,B 0,C 180,E1 5663.847,E2 5663.847} C_VEL
LIN {X 0,Y 113.07,Z 1059.459,A -85,B 0,C 180,E1 5653.033,E2 5653.033} C_VEL
LIN {X 0,Y 116.832,Z 1056.71,A -85,B 0,C 180,E1 5642.474,E2 5642.474} C_VEL
LIN {X 0,Y 123.61,Z 1052.832,A -85,B 0,C 180,E1 5632.651,E2 5632.651} C_VEL
LIN {X 0,Y 134.268,Z 1047.279,A -85,B 0,C 180,E1 5623.131,E2 5623.131} C_VEL
LIN {X 0,Y 149.739,Z 1039.125,A -85,B 0,C 180,E1 5614.105,E2 5614.105} C_VEL
LIN {X 0,Y 164.328,Z 1031.097,A -85,B 0,C 180,E1 5608.082,E2 5608.082} C_VEL
LIN {X 0,Y 181.957,Z 1020.8,A -85,B 0,C 180,E1 5602.604,E2 5602.604} C_VEL
LIN {X 0,Y 200.891,Z 1008.511,A -85,B 0,C 180,E1 5598.075,E2 5598.075} C_VEL
LIN {X 0,Y 217.312,Z 996.91,A -85,B 0,C 180,E1 5594.931,E2 5594.931} C_VEL
LIN {X 0,Y 236.103,Z 982.433,A -85,B 0,C 180,E1 5591.966,E2 5591.966} C_VEL
LIN {X 0,Y 255.019,Z 965.976,A -85,B 0,C 180,E1 5589.478,E2 5589.478} C_VEL
LIN {X 0,Y 270.437,Z 951.242,A -85,B 0,C 180,E1 5587.748,E2 5587.748} C_VEL
LIN {X 0,Y 288.059,Z 932.66,A -85,B 0,C 180,E1 5586.028,E2 5586.028} C_VEL
LIN {X 0,Y 303.968,Z 913.601,A -85,B 0,C 180,E1 5584.658,E2 5584.658} C_VEL
LIN {X 0,Y 317.105,Z 896.169,A -85,B 0,C 180,E1 5583.647,E2 5583.647} C_VEL
LIN {X 0,Y 331.808,Z 874.334,A -85,B 0,C 180,E1 5582.62,E2 5582.62} C_VEL
LIN {X 0,Y 344.135,Z 853.192,A -85,B 0,C 180,E1 5581.83,E2 5581.83} C_VEL
LIN {X 0,Y 354.043,Z 834,A -85,B 0,C 180,E1 5581.25,E2 5581.25} C_VEL
LIN {X 0,Y 364.482,Z 810.876,A -85,B 0,C 180,E1 5580.677,E2 5580.677} C_VEL
LIN {X 0,Y 373.458,Z 786.735,A -85,B 0,C 180,E1 5580.201,E2 5580.201} C_VEL
LIN {X 0,Y 380.238,Z 764.876,A -85,B 0,C 180,E1 5579.874,E2 5579.874} C_VEL
LIN {X 0,Y 386.687,Z 738.841,A -85,B 0,C 180,E1 5579.552,E2 5579.552} C_VEL
LIN {X 0,Y 391.073,Z 713.85,A -85,B 0,C 180,E1 5579.266,E2 5579.266} C_VEL
LIN {X 0,Y 400.495,Z 638.581,A -85,B 0,C 180,E1 5578.419,E2 5578.419} C_VEL
LIN {X 0,Y 390.579,Z 717.226,A -85,B 0,C 180,E1 5577.543,E2 5577.543} C_VEL
LIN {X 0,Y 385.135,Z 745.552,A -85,B 0,C 180,E1 5577.216,E2 5577.216} C_VEL
LIN {X 0,Y 379.415,Z 767.641,A -85,B 0,C 180,E1 5576.915,E2 5576.915} C_VEL
LIN {X 0,Y 372.629,Z 789.081,A -85,B 0,C 180,E1 5576.557,E2 5576.557} C_VEL
LIN {X 0,Y 362.833,Z 814.471,A -85,B 0,C 180,E1 5576.019,E2 5576.019} C_VEL
LIN {X 0,Y 353.177,Z 835.553,A -85,B 0,C 180,E1 5575.453,E2 5575.453} C_VEL
LIN {X 0,Y 342.916,Z 855.184,A -85,B 0,C 180,E1 5574.814,E2 5574.814} C_VEL
LIN {X 0,Y 328.355,Z 879.334,A -85,B 0,C 180,E1 5573.844,E2 5573.844} C_VEL
LIN {X 0,Y 315.86,Z 897.513,A -85,B 0,C 180,E1 5572.937,E2 5572.937} C_VEL
LIN {X 0,Y 301.841,Z 915.873,A -85,B 0,C 180,E1 5571.811,E2 5571.811} C_VEL
LIN {X 0,Y 284.096,Z 936.437,A -85,B 0,C 180,E1 5570.22,E2 5570.22} C_VEL
LIN {X 0,Y 269.185,Z 951.89,A -85,B 0,C 180,E1 5568.702,E2 5568.702} C_VEL
LIN {X 0,Y 253.569,Z 966.642,A -85,B 0,C 180,E1 5566.9,E2 5566.9} C_VEL
LIN {X 0,Y 232.893,Z 984.146,A -85,B 0,C 180,E1 5564.091,E2 5564.091} C_VEL
LIN {X 0,Y 216.292,Z 996.766,A -85,B 0,C 180,E1 5561.384,E2 5561.384} C_VEL
LIN {X 0,Y 198.579,Z 1009.109,A -85,B 0,C 180,E1 5557.892,E2 5557.892} C_VEL
LIN {X 0,Y 179.364,Z 1021.165,A -85,B 0,C 180,E1 5553.117,E2 5553.117} C_VEL
LIN {X 0,Y 163.718,Z 1030.176,A -85,B 0,C 180,E1 5548.094,E2 5548.094} C_VEL
LIN {X 0,Y 148.202,Z 1038.588,A -85,B 0,C 180,E1 5541.501,E2 5541.501} C_VEL
LIN {X 0,Y 133.308,Z 1046.183,A -85,B 0,C 180,E1 5532.458,E2 5532.458} C_VEL
LIN {X 0,Y 123.592,Z 1051.15,A -85,B 0,C 180,E1 5523.561,E2 5523.561} C_VEL
LIN {X 0,Y 116.63,Z 1055.044,A -85,B 0,C 180,E1 5513.226,E2 5513.226} C_VEL
LIN {X 0,Y 112.674,Z 1057.928,A -85,B 0,C 180,E1 5500.74,E2 5500.74} C_VEL
LIN {X 0,Y 111.948,Z 1059.069,A -85,B 0,C 180,E1 5491.023,E2 5491.023} C_VEL
LIN {X 0,Y 111.957,Z 1059.411,A -85,B 0,C 180,E1 5482.817,E2 5482.817} C_VEL
LIN {X 0,Y 112.832,Z 1058.88,A -85,B 0,C 180,E1 5472.464,E2 5472.464} C_VEL
LIN {X 0,Y 116.613,Z 1057.08,A -85,B 0,C 180,E1 5460.998,E2 5460.998} C_VEL
LIN {X 0,Y 123.087,Z 1054.367,A -85,B 0,C 180,E1 5451.247,E2 5451.247} C_VEL
LIN {X 0,Y 133.11,Z 1050.283,A -85,B 0,C 180,E1 5441.955,E2 5441.955} C_VEL
LIN {X 0,Y 149.139,Z 1043.455,A -85,B 0,C 180,E1 5432.354,E2 5432.354} C_VEL
LIN {X 0,Y 164.589,Z 1036.339,A -85,B 0,C 180,E1 5425.959,E2 5425.959} C_VEL
LIN {X 0,Y 181.863,Z 1027.738,A -85,B 0,C 180,E1 5420.602,E2 5420.602} C_VEL
LIN {X 0,Y 202.554,Z 1016.197,A -85,B 0,C 180,E1 5415.72,E2 5415.72} C_VEL
LIN {X 0,Y 219.254,Z 1005.896,A -85,B 0,C 180,E1 5412.597,E2 5412.597} C_VEL
LIN {X 0,Y 237.43,Z 993.61,A -85,B 0,C 180,E1 5409.789,E2 5409.789} C_VEL
LIN {X 0,Y 258.318,Z 977.741,A -85,B 0,C 180,E1 5407.115,E2 5407.115} C_VEL
LIN {X 0,Y 274.18,Z 964.339,A -85,B 0,C 180,E1 5405.388,E2 5405.388} C_VEL
LIN {X 0,Y 291.101,Z 948.617,A -85,B 0,C 180,E1 5403.782,E2 5403.782} C_VEL
LIN {X 0,Y 310.193,Z 928.625,A -85,B 0,C 180,E1 5402.201,E2 5402.201} C_VEL
LIN {X 0,Y 324.406,Z 911.922,A -85,B 0,C 180,E1 5401.158,E2 5401.158} C_VEL
LIN {X 0,Y 337.964,Z 894.276,A -85,B 0,C 180,E1 5400.256,E2 5400.256} C_VEL
LIN {X 0,Y 353.485,Z 871.362,A -85,B 0,C 180,E1 5399.311,E2 5399.311} C_VEL
LIN {X 0,Y 365.058,Z 851.782,A -85,B 0,C 180,E1 5398.659,E2 5398.659} C_VEL
LIN {X 0,Y 366.299,Z 849.549,A -85,B 0,C 180,E1 5398.592,E2 5398.592} C_VEL
LIN {X 0,Y 358.135,Z 863.83,A -85,B 0,C 180,E1 5398.158,E2 5398.158} C_VEL
LIN {X 0,Y 353.391,Z 871.57,A -85,B 0,C 180,E1 5398.06,E2 5398.06} C_VEL
LIN {X 0,Y 340.493,Z 890.789,A -85,B 0,C 180,E1 5398.353,E2 5398.353} C_VEL
LIN {X 0,Y 335.246,Z 897.809,A -85,B 0,C 180,E1 5398.223,E2 5398.223} C_VEL
LIN {X 0,Y 321.3,Z 915.55,A -85,B 0,C 180,E1 5397.377,E2 5397.377} C_VEL
LIN {X 0,Y 302.178,Z 937.044,A -85,B 0,C 180,E1 5396.064,E2 5396.064} C_VEL
LIN {X 0,Y 286.14,Z 953.042,A -85,B 0,C 180,E1 5394.811,E2 5394.811} C_VEL
LIN {X 0,Y 267.871,Z 969.526,A -85,B 0,C 180,E1 5393.169,E2 5393.169} C_VEL
LIN {X 0,Y 247.976,Z 985.399,A -85,B 0,C 180,E1 5391.073,E2 5391.073} C_VEL
LIN {X 0,Y 231.233,Z 997.456,A -85,B 0,C 180,E1 5388.986,E2 5388.986} C_VEL
LIN {X 0,Y 213.051,Z 1009.373,A -85,B 0,C 180,E1 5386.285,E2 5386.285} C_VEL
LIN {X 0,Y 191.118,Z 1022.196,A -85,B 0,C 180,E1 5382.21,E2 5382.21} C_VEL
LIN {X 0,Y 173.506,Z 1031.403,A -85,B 0,C 180,E1 5378.001,E2 5378.001} C_VEL
LIN {X 0,Y 155.665,Z 1039.927,A -85,B 0,C 180,E1 5372.427,E2 5372.427} C_VEL
LIN {X 0,Y 137.17,Z 1047.857,A -85,B 0,C 180,E1 5364.327,E2 5364.327} C_VEL
LIN {X 0,Y 124.045,Z 1053.098,A -85,B 0,C 180,E1 5355.84,E2 5355.84} C_VEL
LIN {X 0,Y 112.94,Z 1057.495,A -85,B 0,C 180,E1 5344.514,E2 5344.514} C_VEL
LIN {X 0,Y 106.261,Z 1060.174,A -85,B 0,C 180,E1 5331.53,E2 5331.53} C_VEL
LIN {X 0,Y 104.143,Z 1061.244,A -85,B 0,C 180,E1 5320.511,E2 5320.511} C_VEL
LIN {X 0,Y 103.909,Z 1061.41,A -85,B 0,C 180,E1 5311.654,E2 5311.654} C_VEL
LIN {X 0,Y 103.929,Z 1061.073,A -85,B 0,C 180,E1 5303.925,E2 5303.925} C_VEL
LIN {X 0,Y 105.179,Z 1059.472,A -85,B 0,C 180,E1 5292.29,E2 5292.29} C_VEL
LIN {X 0,Y 109.606,Z 1056.596,A -85,B 0,C 180,E1 5280.488,E2 5280.488} C_VEL
LIN {X 0,Y 117.133,Z 1052.707,A -85,B 0,C 180,E1 5270.192,E2 5270.192} C_VEL
LIN {X 0,Y 128.72,Z 1047.143,A -85,B 0,C 180,E1 5260.426,E2 5260.426} C_VEL
LIN {X 0,Y 145.22,Z 1038.968,A -85,B 0,C 180,E1 5251.375,E2 5251.375} C_VEL
LIN {X 0,Y 160.589,Z 1030.917,A -85,B 0,C 180,E1 5245.444,E2 5245.444} C_VEL
LIN {X 0,Y 179.736,Z 1020.141,A -85,B 0,C 180,E1 5239.923,E2 5239.923} C_VEL
LIN {X 0,Y 199.331,Z 1007.725,A -85,B 0,C 180,E1 5235.611,E2 5235.611} C_VEL
LIN {X 0,Y 216.216,Z 996.049,A -85,B 0,C 180,E1 5232.641,E2 5232.641} C_VEL
LIN {X 0,Y 236.374,Z 980.649,A -85,B 0,C 180,E1 5229.732,E2 5229.732} C_VEL
LIN {X 0,Y 254.194,Z 965.341,A -85,B 0,C 180,E1 5227.585,E2 5227.585} C_VEL
LIN {X 0,Y 270.405,Z 950.024,A -85,B 0,C 180,E1 5225.91,E2 5225.91} C_VEL
LIN {X 0,Y 289.738,Z 929.531,A -85,B 0,C 180,E1 5224.183,E2 5224.183} C_VEL
LIN {X 0,Y 304.391,Z 912.028,A -85,B 0,C 180,E1 5223.034,E2 5223.034} C_VEL
LIN {X 0,Y 318.169,Z 893.778,A -85,B 0,C 180,E1 5222.067,E2 5222.067} C_VEL
LIN {X 0,Y 333.521,Z 870.628,A -85,B 0,C 180,E1 5221.086,E2 5221.086} C_VEL
LIN {X 0,Y 344.47,Z 851.818,A -85,B 0,C 180,E1 5220.442,E2 5220.442} C_VEL
LIN {X 0,Y 354.959,Z 831.461,A -85,B 0,C 180,E1 5219.879,E2 5219.879} C_VEL
LIN {X 0,Y 366.318,Z 805.553,A -85,B 0,C 180,E1 5219.308,E2 5219.308} C_VEL
LIN {X 0,Y 374.02,Z 784.534,A -85,B 0,C 180,E1 5218.936,E2 5218.936} C_VEL
LIN {X 0,Y 380.998,Z 761.779,A -85,B 0,C 180,E1 5218.624,E2 5218.624} C_VEL
LIN {X 0,Y 385.322,Z 744.469,A -85,B 0,C 180,E1 5218.421,E2 5218.421} C_VEL
LIN {X 0,Y 379.469,Z 767.072,A -85,B 0,C 180,E1 5218.135,E2 5218.135} C_VEL
LIN {X 0,Y 372.729,Z 788.325,A -85,B 0,C 180,E1 5217.808,E2 5217.808} C_VEL
LIN {X 0,Y 362.366,Z 815.032,A -85,B 0,C 180,E1 5217.279,E2 5217.279} C_VEL
LIN {X 0,Y 352.627,Z 836.072,A -85,B 0,C 180,E1 5216.749,E2 5216.749} C_VEL
LIN {X 0,Y 341.255,Z 857.524,A -85,B 0,C 180,E1 5216.088,E2 5216.088} C_VEL
LIN {X 0,Y 327.59,Z 879.729,A -85,B 0,C 180,E1 5215.243,E2 5215.243} C_VEL
LIN {X 0,Y 314.97,Z 897.879,A -85,B 0,C 180,E1 5214.392,E2 5214.392} C_VEL
LIN {X 0,Y 300.529,Z 916.549,A -85,B 0,C 180,E1 5213.313,E2 5213.313} C_VEL
LIN {X 0,Y 282.832,Z 936.735,A -85,B 0,C 180,E1 5211.837,E2 5211.837} C_VEL
LIN {X 0,Y 267.712,Z 952.17,A -85,B 0,C 180,E1 5210.408,E2 5210.408} C_VEL
LIN {X 0,Y 250.923,Z 967.74,A -85,B 0,C 180,E1 5208.598,E2 5208.598} C_VEL
LIN {X 0,Y 230.788,Z 984.38,A -85,B 0,C 180,E1 5206.042,E2 5206.042} C_VEL
LIN {X 0,Y 213.821,Z 996.987,A -85,B 0,C 180,E1 5203.462,E2 5203.462} C_VEL
LIN {X 0,Y 194.795,Z 1009.882,A -85,B 0,C 180,E1 5199.94,E2 5199.94} C_VEL
LIN {X 0,Y 175.007,Z 1021.8,A -85,B 0,C 180,E1 5195.289,E2 5195.289} C_VEL
LIN {X 0,Y 158.789,Z 1030.745,A -85,B 0,C 180,E1 5190.34,E2 5190.34} C_VEL
LIN {X 0,Y 141.261,Z 1039.749,A -85,B 0,C 180,E1 5183.115,E2 5183.115} C_VEL
LIN {X 0,Y 126.85,Z 1046.569,A -85,B 0,C 180,E1 5174.55,E2 5174.55} C_VEL
LIN {X 0,Y 116.577,Z 1051.426,A -85,B 0,C 180,E1 5165.43,E2 5165.43} C_VEL
LIN {X 0,Y 108.464,Z 1055.63,A -85,B 0,C 180,E1 5153.353,E2 5153.353} C_VEL
LIN {X 0,Y 104.605,Z 1058.155,A -85,B 0,C 180,E1 5140.464,E2 5140.464} C_VEL
LIN {X 0,Y 103.952,Z 1059.174,A -85,B 0,C 180,E1 5130.551,E2 5130.551} C_VEL
LIN {X 0,Y 103.961,Z 1059.48,A -85,B 0,C 180,E1 5122.162,E2 5122.162} C_VEL
LIN {X 0,Y 105.054,Z 1058.944,A -85,B 0,C 180,E1 5111.119,E2 5111.119} C_VEL
LIN {X 0,Y 109.282,Z 1057.197,A -85,B 0,C 180,E1 5099.177,E2 5099.177} C_VEL
LIN {X 0,Y 116.661,Z 1054.421,A -85,B 0,C 180,E1 5088.703,E2 5088.703} C_VEL
LIN {X 0,Y 127.645,Z 1050.317,A -85,B 0,C 180,E1 5079.149,E2 5079.149} C_VEL
LIN {X 0,Y 144.803,Z 1043.468,A -85,B 0,C 180,E1 5069.536,E2 5069.536} C_VEL
LIN {X 0,Y 160.295,Z 1036.694,A -85,B 0,C 180,E1 5063.515,E2 5063.515} C_VEL
LIN {X 0,Y 177.186,Z 1028.641,A -85,B 0,C 180,E1 5058.55,E2 5058.55} C_VEL
LIN {X 0,Y 199.55,Z 1016.677,A -85,B 0,C 180,E1 5053.572,E2 5053.572} C_VEL
LIN {X 0,Y 217.575,Z 1005.848,A -85,B 0,C 180,E1 5050.437,E2 5050.437} C_VEL
LIN {X 0,Y 237.09,Z 992.911,A -85,B 0,C 180,E1 5047.663,E2 5047.663} C_VEL
LIN {X 0,Y 257.072,Z 977.928,A -85,B 0,C 180,E1 5045.306,E2 5045.306} C_VEL
LIN {X 0,Y 273.523,Z 964.232,A -85,B 0,C 180,E1 5043.65,E2 5043.65} C_VEL
LIN {X 0,Y 290.393,Z 948.754,A -85,B 0,C 180,E1 5042.171,E2 5042.171} C_VEL
LIN {X 0,Y 309.438,Z 929.075,A -85,B 0,C 180,E1 5040.711,E2 5040.711} C_VEL
LIN {X 0,Y 323.966,Z 912.196,A -85,B 0,C 180,E1 5039.724,E2 5039.724} C_VEL
LIN {X 0,Y 337.302,Z 895.032,A -85,B 0,C 180,E1 5038.905,E2 5038.905} C_VEL
LIN {X 0,Y 342.061,Z 888.504,A -85,B 0,C 180,E1 5038.612,E2 5038.612} C_VEL
LIN {X 0,Y 335.246,Z 897.809,A -85,B 0,C 180,E1 5038.223,E2 5038.223} C_VEL
LIN {X 0,Y 330.034,Z 904.784,A -85,B 0,C 180,E1 5038.089,E2 5038.089} C_VEL
LIN {X 0,Y 315.837,Z 921.858,A -85,B 0,C 180,E1 5038.328,E2 5038.328} C_VEL
LIN {X 0,Y 310.178,Z 928.13,A -85,B 0,C 180,E1 5038.16,E2 5038.16} C_VEL
LIN {X 0,Y 292.381,Z 946.71,A -85,B 0,C 180,E1 5036.95,E2 5036.95} C_VEL
LIN {X 0,Y 273.81,Z 963.738,A -85,B 0,C 180,E1 5035.508,E2 5035.508} C_VEL
LIN {X 0,Y 257.365,Z 977.388,A -85,B 0,C 180,E1 5034.033,E2 5034.033} C_VEL
LIN {X 0,Y 237.333,Z 992.442,A -85,B 0,C 180,E1 5031.914,E2 5031.914} C_VEL
LIN {X 0,Y 216.757,Z 1005.987,A -85,B 0,C 180,E1 5029.282,E2 5029.282} C_VEL
LIN {X 0,Y 198.528,Z 1016.827,A -85,B 0,C 180,E1 5026.42,E2 5026.42} C_VEL
LIN {X 0,Y 177.448,Z 1028.124,A -85,B 0,C 180,E1 5022.229,E2 5022.229} C_VEL
LIN {X 0,Y 157.518,Z 1037.447,A -85,B 0,C 180,E1 5016.989,E2 5016.989} C_VEL
LIN {X 0,Y 141.273,Z 1044.357,A -85,B 0,C 180,E1 5011.23,E2 5011.23} C_VEL
LIN {X 0,Y 123.748,Z 1051.189,A -85,B 0,C 180,E1 5002.358,E2 5002.358} C_VEL
LIN {X 0,Y 110.606,Z 1055.834,A -85,B 0,C 180,E1 4991.987,E2 4991.987} C_VEL
LIN {X 0,Y 102.313,Z 1058.757,A -85,B 0,C 180,E1 4981.196,E2 4981.196} C_VEL
LIN {X 0,Y 97.486,Z 1060.598,A -85,B 0,C 180,E1 4969.161,E2 4969.161} C_VEL
LIN {X 0,Y 95.963,Z 1061.339,A -85,B 0,C 180,E1 4957.183,E2 4957.183} C_VEL
LIN {X 0,Y 95.915,Z 1061.215,A -85,B 0,C 180,E1 4948.806,E2 4948.806} C_VEL
LIN {X 0,Y 96.075,Z 1060.636,A -85,B 0,C 180,E1 4940.415,E2 4940.415} C_VEL
LIN {X 0,Y 97.914,Z 1059.021,A -85,B 0,C 180,E1 4929.059,E2 4929.059} C_VEL
LIN {X 0,Y 102.848,Z 1056.32,A -85,B 0,C 180,E1 4917.676,E2 4917.676} C_VEL
LIN {X 0,Y 111.373,Z 1052.372,A -85,B 0,C 180,E1 4906.976,E2 4906.976} C_VEL
LIN {X 0,Y 125.357,Z 1046.206,A -85,B 0,C 180,E1 4896.332,E2 4896.332} C_VEL
LIN {X 0,Y 141.786,Z 1038.453,A -85,B 0,C 180,E1 4888.176,E2 4888.176} C_VEL
LIN {X 0,Y 157.959,Z 1030.35,A -85,B 0,C 180,E1 4882.455,E2 4882.455} C_VEL
LIN {X 0,Y 178.776,Z 1018.908,A -85,B 0,C 180,E1 4876.983,E2 4876.983} C_VEL
LIN {X 0,Y 197.248,Z 1007.521,A -85,B 0,C 180,E1 4873.275,E2 4873.275} C_VEL
LIN {X 0,Y 214.546,Z 995.83,A -85,B 0,C 180,E1 4870.468,E2 4870.468} C_VEL
LIN {X 0,Y 236.058,Z 979.62,A -85,B 0,C 180,E1 4867.622,E2 4867.622} C_VEL
LIN {X 0,Y 253.233,Z 965.077,A -85,B 0,C 180,E1 4865.725,E2 4865.725} C_VEL
LIN {X 0,Y 269.679,Z 949.742,A -85,B 0,C 180,E1 4864.161,E2 4864.161} C_VEL
LIN {X 0,Y 289.253,Z 929.211,A -85,B 0,C 180,E1 4862.553,E2 4862.553} C_VEL
LIN {X 0,Y 303.709,Z 912.128,A -85,B 0,C 180,E1 4861.509,E2 4861.509} C_VEL
LIN {X 0,Y 317.979,Z 893.41,A -85,B 0,C 180,E1 4860.589,E2 4860.589} C_VEL
LIN {X 0,Y 332.965,Z 871.02,A -85,B 0,C 180,E1 4859.71,E2 4859.71} C_VEL
LIN {X 0,Y 344.475,Z 851.404,A -85,B 0,C 180,E1 4859.087,E2 4859.087} C_VEL
LIN {X 0,Y 355.573,Z 829.939,A -85,B 0,C 180,E1 4858.54,E2 4858.54} C_VEL
LIN {X 0,Y 358.843,Z 822.891,A -85,B 0,C 180,E1 4858.381,E2 4858.381} C_VEL
LIN {X 0,Y 346.23,Z 848.184,A -85,B 0,C 180,E1 4857.735,E2 4857.735} C_VEL
LIN {X 0,Y 334.838,Z 867.866,A -85,B 0,C 180,E1 4857.105,E2 4857.105} C_VEL
LIN {X 0,Y 321.628,Z 888.125,A -85,B 0,C 180,E1 4856.314,E2 4856.314} C_VEL
LIN {X 0,Y 305.509,Z 909.687,A -85,B 0,C 180,E1 4855.259,E2 4855.259} C_VEL
LIN {X 0,Y 291.439,Z 926.452,A -85,B 0,C 180,E1 4854.237,E2 4854.237} C_VEL
LIN {X 0,Y 275.012,Z 944.119,A -85,B 0,C 180,E1 4852.899,E2 4852.899} C_VEL
LIN {X 0,Y 256.035,Z 962.154,A -85,B 0,C 180,E1 4851.125,E2 4851.125} C_VEL
LIN {X 0,Y 239.143,Z 976.568,A -85,B 0,C 180,E1 4849.283,E2 4849.283} C_VEL
LIN {X 0,Y 219.792,Z 991.536,A -85,B 0,C 180,E1 4846.788,E2 4846.788} C_VEL
LIN {X 0,Y 200.029,Z 1004.995,A -85,B 0,C 180,E1 4843.688,E2 4843.688} C_VEL
LIN {X 0,Y 182.656,Z 1015.739,A -85,B 0,C 180,E1 4840.313,E2 4840.313} C_VEL
LIN {X 0,Y 162.789,Z 1026.923,A -85,B 0,C 180,E1 4835.373,E2 4835.373} C_VEL
LIN {X 0,Y 144.331,Z 1036.12,A -85,B 0,C 180,E1 4829.208,E2 4829.208} C_VEL
LIN {X 0,Y 129.762,Z 1042.893,A -85,B 0,C 180,E1 4822.501,E2 4822.501} C_VEL
LIN {X 0,Y 114.587,Z 1049.641,A -85,B 0,C 180,E1 4812.214,E2 4812.214} C_VEL
LIN {X 0,Y 104.177,Z 1054.175,A -85,B 0,C 180,E1 4800.576,E2 4800.576} C_VEL
LIN {X 0,Y 98.728,Z 1056.899,A -85,B 0,C 180,E1 4789.524,E2 4789.524} C_VEL
LIN {X 0,Y 96.386,Z 1058.514,A -85,B 0,C 180,E1 4778.952,E2 4778.952} C_VEL
LIN {X 0,Y 95.94,Z 1059.279,A -85,B 0,C 180,E1 4770,E2 4770} C_VEL
LIN {X 0,Y 95.988,Z 1059.536,A -85,B 0,C 180,E1 4761.01,E2 4761.01} C_VEL
LIN {X 0,Y 97.474,Z 1058.942,A -85,B 0,C 180,E1 4748.959,E2 4748.959} C_VEL
LIN {X 0,Y 102.233,Z 1057.252,A -85,B 0,C 180,E1 4736.79,E2 4736.79} C_VEL
LIN {X 0,Y 110.514,Z 1054.466,A -85,B 0,C 180,E1 4725.84,E2 4725.84} C_VEL
LIN {X 0,Y 123.127,Z 1050.146,A -85,B 0,C 180,E1 4715.701,E2 4715.701} C_VEL
LIN {X 0,Y 140.838,Z 1043.48,A -85,B 0,C 180,E1 4706.55,E2 4706.55} C_VEL
LIN {X 0,Y 157.924,Z 1036.342,A -85,B 0,C 180,E1 4700.437,E2 4700.437} C_VEL
LIN {X 0,Y 178.151,Z 1027.007,A -85,B 0,C 180,E1 4695.124,E2 4695.124} C_VEL
LIN {X 0,Y 198.747,Z 1016.073,A -85,B 0,C 180,E1 4691.022,E2 4691.022} C_VEL
LIN {X 0,Y 216.242,Z 1005.782,A -85,B 0,C 180,E1 4688.241,E2 4688.241} C_VEL
LIN {X 0,Y 236.724,Z 992.448,A -85,B 0,C 180,E1 4685.575,E2 4685.575} C_VEL
LIN {X 0,Y 257.41,Z 977.063,A -85,B 0,C 180,E1 4683.349,E2 4683.349} C_VEL
LIN {X 0,Y 274.107,Z 963.274,A -85,B 0,C 180,E1 4681.823,E2 4681.823} C_VEL
LIN {X 0,Y 292.971,Z 946.032,A -85,B 0,C 180,E1 4680.331,E2 4680.331} C_VEL
LIN {X 0,Y 310.552,Z 927.681,A -85,B 0,C 180,E1 4679.107,E2 4679.107} C_VEL
LIN {X 0,Y 317.875,Z 919.553,A -85,B 0,C 180,E1 4678.634,E2 4678.634} C_VEL
LIN {X 0,Y 310.178,Z 928.13,A -85,B 0,C 180,E1 4678.16,E2 4678.16} C_VEL
LIN {X 0,Y 304.963,Z 933.856,A -85,B 0,C 180,E1 4678.013,E2 4678.013} C_VEL
LIN {X 0,Y 290.734,Z 948.093,A -85,B 0,C 180,E1 4678.265,E2 4678.265} C_VEL
LIN {X 0,Y 285.126,Z 953.28,A -85,B 0,C 180,E1 4678.088,E2 4678.088} C_VEL
LIN {X 0,Y 266.417,Z 969.73,A -85,B 0,C 180,E1 4676.678,E2 4676.678} C_VEL
LIN {X 0,Y 245.932,Z 985.559,A -85,B 0,C 180,E1 4674.868,E2 4674.868} C_VEL
LIN {X 0,Y 228.65,Z 997.571,A -85,B 0,C 180,E1 4673.058,E2 4673.058} C_VEL
LIN {X 0,Y 208.804,Z 1010.033,A -85,B 0,C 180,E1 4670.561,E2 4670.561} C_VEL
LIN {X 0,Y 186.058,Z 1022.565,A -85,B 0,C 180,E1 4666.955,E2 4666.955} C_VEL
LIN {X 0,Y 168.076,Z 1031.371,A -85,B 0,C 180,E1 4663.293,E2 4663.293} C_VEL
LIN {X 0,Y 148.686,Z 1039.916,A -85,B 0,C 180,E1 4658.129,E2 4658.129} C_VEL
LIN {X 0,Y 128.585,Z 1047.662,A -85,B 0,C 180,E1 4650.566,E2 4650.566} C_VEL
LIN {X 0,Y 113.736,Z 1052.817,A -85,B 0,C 180,E1 4642.299,E2 4642.299} C_VEL
LIN {X 0,Y 100.687,Z 1057.079,A -85,B 0,C 180,E1 4630.952,E2 4630.952} C_VEL
LIN {X 0,Y 91.489,Z 1059.974,A -85,B 0,C 180,E1 4615.923,E2 4615.923} C_VEL
LIN {X 0,Y 88.358,Z 1061.072,A -85,B 0,C 180,E1 4603.081,E2 4603.081} C_VEL
LIN {X 0,Y 87.905,Z 1061.267,A -85,B 0,C 180,E1 4592.608,E2 4592.608} C_VEL
LIN {X 0,Y 87.923,Z 1060.971,A -85,B 0,C 180,E1 4584.126,E2 4584.126} C_VEL
LIN {X 0,Y 89.316,Z 1059.614,A -85,B 0,C 180,E1 4571.056,E2 4571.056} C_VEL
LIN {X 0,Y 95.266,Z 1056.531,A -85,B 0,C 180,E1 4556.202,E2 4556.202} C_VEL
LIN {X 0,Y 104.42,Z 1052.669,A -85,B 0,C 180,E1 4544.88,E2 4544.88} C_VEL
LIN {X 0,Y 117.947,Z 1047.132,A -85,B 0,C 180,E1 4534.684,E2 4534.684} C_VEL
LIN {X 0,Y 136.501,Z 1039.013,A -85,B 0,C 180,E1 4525.712,E2 4525.712} C_VEL
LIN {X 0,Y 153.294,Z 1031.004,A -85,B 0,C 180,E1 4520.073,E2 4520.073} C_VEL
LIN {X 0,Y 172.103,Z 1021.191,A -85,B 0,C 180,E1 4515.329,E2 4515.329} C_VEL
LIN {X 0,Y 193.664,Z 1008.476,A -85,B 0,C 180,E1 4511.197,E2 4511.197} C_VEL
LIN {X 0,Y 211.307,Z 996.897,A -85,B 0,C 180,E1 4508.521,E2 4508.521} C_VEL
LIN {X 0,Y 231.256,Z 982.443,A -85,B 0,C 180,E1 4506.039,E2 4506.039} C_VEL
LIN {X 0,Y 250.591,Z 966.523,A -85,B 0,C 180,E1 4504.035,E2 4504.035} C_VEL
LIN {X 0,Y 267.106,Z 951.458,A -85,B 0,C 180,E1 4502.575,E2 4502.575} C_VEL
LIN {X 0,Y 285.525,Z 932.82,A -85,B 0,C 180,E1 4501.167,E2 4501.167} C_VEL
LIN {X 0,Y 302.514,Z 913.126,A -85,B 0,C 180,E1 4500.025,E2 4500.025} C_VEL
LIN {X 0,Y 315.992,Z 895.743,A -85,B 0,C 180,E1 4499.224,E2 4499.224} C_VEL
LIN {X 0,Y 331.089,Z 873.87,A -85,B 0,C 180,E1 4498.407,E2 4498.407} C_VEL
LIN {X 0,Y 332.098,Z 872.229,A -85,B 0,C 180,E1 4498.351,E2 4498.351} C_VEL
LIN {X 0,Y 316.766,Z 894.643,A -85,B 0,C 180,E1 4497.494,E2 4497.494} C_VEL
LIN {X 0,Y 302.984,Z 912.437,A -85,B 0,C 180,E1 4496.645,E2 4496.645} C_VEL
LIN {X 0,Y 287.322,Z 930.616,A -85,B 0,C 180,E1 4495.577,E2 4495.577} C_VEL
LIN {X 0,Y 268.383,Z 949.983,A -85,B 0,C 180,E1 4494.115,E2 4494.115} C_VEL
LIN {X 0,Y 252.035,Z 964.924,A -85,B 0,C 180,E1 4492.662,E2 4492.662} C_VEL
LIN {X 0,Y 233.041,Z 980.624,A -85,B 0,C 180,E1 4490.691,E2 4490.691} C_VEL
LIN {X 0,Y 212.512,Z 995.542,A -85,B 0,C 180,E1 4488.139,E2 4488.139} C_VEL
LIN {X 0,Y 195.177,Z 1006.898,A -85,B 0,C 180,E1 4485.521,E2 4485.521} C_VEL
LIN {X 0,Y 174.649,Z 1019.085,A -85,B 0,C 180,E1 4481.646,E2 4481.646} C_VEL
LIN {X 0,Y 154.593,Z 1029.489,A -85,B 0,C 180,E1 4476.698,E2 4476.698} C_VEL
LIN {X 0,Y 138.022,Z 1037.323,A -85,B 0,C 180,E1 4471.231,E2 4471.231} C_VEL
LIN {X 0,Y 120.251,Z 1045.09,A -85,B 0,C 180,E1 4462.962,E2 4462.962} C_VEL
LIN {X 0,Y 105.399,Z 1051.004,A -85,B 0,C 180,E1 4452.271,E2 4452.271} C_VEL
LIN {X 0,Y 95.777,Z 1054.916,A -85,B 0,C 180,E1 4440.767,E2 4440.767} C_VEL
LIN {X 0,Y 89.641,Z 1057.895,A -85,B 0,C 180,E1 4426.192,E2 4426.192} C_VEL
LIN {X 0,Y 87.978,Z 1059.251,A -85,B 0,C 180,E1 4413.257,E2 4413.257} C_VEL
LIN {X 0,Y 87.927,Z 1059.569,A -85,B 0,C 180,E1 4404.125,E2 4404.125} C_VEL
LIN {X 0,Y 88.65,Z 1059.375,A -85,B 0,C 180,E1 4392.947,E2 4392.947} C_VEL
LIN {X 0,Y 93.418,Z 1057.979,A -85,B 0,C 180,E1 4377.644,E2 4377.644} C_VEL
LIN {X 0,Y 103.135,Z 1054.985,A -85,B 0,C 180,E1 4364.158,E2 4364.158} C_VEL
LIN {X 0,Y 115.36,Z 1051.142,A -85,B 0,C 180,E1 4354.291,E2 4354.291} C_VEL
LIN {X 0,Y 132.668,Z 1045.266,A -85,B 0,C 180,E1 4345.256,E2 4345.256} C_VEL
LIN {X 0,Y 152.652,Z 1037.403,A -85,B 0,C 180,E1 4338.238,E2 4338.238} C_VEL
LIN {X 0,Y 169.897,Z 1029.838,A -85,B 0,C 180,E1 4333.816,E2 4333.816} C_VEL
LIN {X 0,Y 191.639,Z 1019.187,A -85,B 0,C 180,E1 4329.559,E2 4329.559} C_VEL
LIN {X 0,Y 212.304,Z 1007.481,A -85,B 0,C 180,E1 4326.412,E2 4326.412} C_VEL
LIN {X 0,Y 229.744,Z 996.527,A -85,B 0,C 180,E1 4324.243,E2 4324.243} C_VEL
LIN {X 0,Y 250.144,Z 982.313,A -85,B 0,C 180,E1 4322.128,E2 4322.128} C_VEL
LIN {X 0,Y 269.975,Z 966.568,A -85,B 0,C 180,E1 4320.395,E2 4320.395} C_VEL
LIN {X 0,Y 287.001,Z 951.503,A -85,B 0,C 180,E1 4319.115,E2 4319.115} C_VEL
LIN {X 0,Y 293.7,Z 945.232,A -85,B 0,C 180,E1 4318.661,E2 4318.661} C_VEL
LIN {X 0,Y 285.126,Z 953.28,A -85,B 0,C 180,E1 4318.088,E2 4318.088} C_VEL
LIN {X 0,Y 279.419,Z 958.574,A -85,B 0,C 180,E1 4317.895,E2 4317.895} C_VEL
LIN {X 0,Y 263.156,Z 972.186,A -85,B 0,C 180,E1 4318.065,E2 4318.065} C_VEL
LIN {X 0,Y 257.988,Z 976.152,A -85,B 0,C 180,E1 4317.841,E2 4317.841} C_VEL
LIN {X 0,Y 239.482,Z 989.799,A -85,B 0,C 180,E1 4316.263,E2 4316.263} C_VEL
LIN {X 0,Y 216.215,Z 1004.931,A -85,B 0,C 180,E1 4313.863,E2 4313.863} C_VEL
LIN {X 0,Y 197.178,Z 1015.862,A -85,B 0,C 180,E1 4311.432,E2 4311.432} C_VEL
LIN {X 0,Y 176.74,Z 1026.378,A -85,B 0,C 180,E1 4308.161,E2 4308.161} C_VEL
LIN {X 0,Y 154.39,Z 1036.377,A -85,B 0,C 180,E1 4303.436,E2 4303.436} C_VEL
LIN {X 0,Y 135.805,Z 1043.672,A -85,B 0,C 180,E1 4298.078,E2 4298.078} C_VEL
LIN {X 0,Y 116.512,Z 1050.445,A -85,B 0,C 180,E1 4290.085,E2 4290.085} C_VEL
LIN {X 0,Y 99.503,Z 1055.58,A -85,B 0,C 180,E1 4278.909,E2 4278.909} C_VEL
LIN {X 0,Y 88.65,Z 1058.645,A -85,B 0,C 180,E1 4266.712,E2 4266.712} C_VEL
LIN {X 0,Y 82.044,Z 1060.543,A -85,B 0,C 180,E1 4252.145,E2 4252.145} C_VEL
LIN {X 0,Y 79.958,Z 1061.239,A -85,B 0,C 180,E1 4237.184,E2 4237.184} C_VEL
LIN {X 0,Y 79.907,Z 1061.028,A -85,B 0,C 180,E1 4227.849,E2 4227.849} C_VEL
LIN {X 0,Y 80.24,Z 1060.381,A -85,B 0,C 180,E1 4217.77,E2 4217.77} C_VEL
LIN {X 0,Y 83.096,Z 1058.699,A -85,B 0,C 180,E1 4204.331,E2 4204.331} C_VEL
LIN {X 0,Y 90.207,Z 1055.766,A -85,B 0,C 180,E1 4190.817,E2 4190.817} C_VEL
LIN {X 0,Y 103.492,Z 1050.86,A -85,B 0,C 180,E1 4177.605,E2 4177.605} C_VEL
LIN {X 0,Y 120.658,Z 1044.065,A -85,B 0,C 180,E1 4167.539,E2 4167.539} C_VEL
LIN {X 0,Y 137.156,Z 1037.062,A -85,B 0,C 180,E1 4161.072,E2 4161.072} C_VEL
LIN {X 0,Y 157.594,Z 1027.524,A -85,B 0,C 180,E1 4155.337,E2 4155.337} C_VEL
LIN {X 0,Y 178.291,Z 1016.434,A -85,B 0,C 180,E1 4151.06,E2 4151.06} C_VEL
LIN {X 0,Y 195.981,Z 1005.945,A -85,B 0,C 180,E1 4148.2,E2 4148.2} C_VEL
LIN {X 0,Y 216.962,Z 992.144,A -85,B 0,C 180,E1 4145.469,E2 4145.469} C_VEL
LIN {X 0,Y 236.435,Z 977.525,A -85,B 0,C 180,E1 4143.394,E2 4143.394} C_VEL
LIN {X 0,Y 253.108,Z 963.693,A -85,B 0,C 180,E1 4141.892,E2 4141.892} C_VEL
LIN {X 0,Y 272.147,Z 946.203,A -85,B 0,C 180,E1 4140.421,E2 4140.421} C_VEL
LIN {X 0,Y 289.992,Z 927.448,A -85,B 0,C 180,E1 4139.223,E2 4139.223} C_VEL
LIN {X 0,Y 304.59,Z 910.384,A -85,B 0,C 180,E1 4138.356,E2 4138.356} C_VEL
LIN {X 0,Y 305.096,Z 909.767,A -85,B 0,C 180,E1 4138.317,E2 4138.317} C_VEL
LIN {X 0,Y 290.543,Z 926.775,A -85,B 0,C 180,E1 4137.436,E2 4137.436} C_VEL
LIN {X 0,Y 273.545,Z 944.651,A -85,B 0,C 180,E1 4136.277,E2 4136.277} C_VEL
LIN {X 0,Y 254.035,Z 962.679,A -85,B 0,C 180,E1 4134.752,E2 4134.752} C_VEL
LIN {X 0,Y 237.268,Z 976.576,A -85,B 0,C 180,E1 4133.223,E2 4133.223} C_VEL
LIN {X 0,Y 217.589,Z 991.309,A -85,B 0,C 180,E1 4131.11,E2 4131.11} C_VEL
LIN {X 0,Y 196.986,Z 1004.838,A -85,B 0,C 180,E1 4128.421,E2 4128.421} C_VEL
LIN {X 0,Y 178.704,Z 1015.617,A -85,B 0,C 180,E1 4125.458,E2 4125.458} C_VEL
LIN {X 0,Y 157.523,Z 1026.859,A -85,B 0,C 180,E1 4121.046,E2 4121.046} C_VEL
LIN {X 0,Y 137.469,Z 1036.089,A -85,B 0,C 180,E1 4115.393,E2 4115.393} C_VEL
LIN {X 0,Y 120.517,Z 1043.176,A -85,B 0,C 180,E1 4108.71,E2 4108.71} C_VEL
LIN {X 0,Y 103.072,Z 1049.892,A -85,B 0,C 180,E1 4098.327,E2 4098.327} C_VEL
LIN {X 0,Y 90.554,Z 1054.404,A -85,B 0,C 180,E1 4085.818,E2 4085.818} C_VEL
LIN {X 0,Y 83.413,Z 1057.218,A -85,B 0,C 180,E1 4072.556,E2 4072.556} C_VEL
LIN {X 0,Y 80.386,Z 1058.834,A -85,B 0,C 180,E1 4059.305,E2 4059.305} C_VEL
LIN {X 0,Y 79.92,Z 1059.467,A -85,B 0,C 180,E1 4049.283,E2 4049.283} C_VEL
LIN {X 0,Y 80.021,Z 1059.705,A -85,B 0,C 180,E1 4039.925,E2 4039.925} C_VEL
LIN {X 0,Y 82.344,Z 1059.071,A -85,B 0,C 180,E1 4024.849,E2 4024.849} C_VEL
LIN {X 0,Y 88.787,Z 1057.362,A -85,B 0,C 180,E1 4010.902,E2 4010.902} C_VEL
LIN {X 0,Y 99.188,Z 1054.556,A -85,B 0,C 180,E1 3999.084,E2 3999.084} C_VEL
LIN {X 0,Y 114.841,Z 1050.01,A -85,B 0,C 180,E1 3988.433,E2 3988.433} C_VEL
LIN {X 0,Y 134.965,Z 1043.203,A -85,B 0,C 180,E1 3979.8,E2 3979.8} C_VEL
LIN {X 0,Y 152.85,Z 1036.345,A -85,B 0,C 180,E1 3974.497,E2 3974.497} C_VEL
LIN {X 0,Y 174.511,Z 1026.984,A -85,B 0,C 180,E1 3969.77,E2 3969.77} C_VEL
LIN {X 0,Y 196.584,Z 1015.81,A -85,B 0,C 180,E1 3966.132,E2 3966.132} C_VEL
LIN {X 0,Y 215.419,Z 1005.132,A -85,B 0,C 180,E1 3963.678,E2 3963.678} C_VEL
LIN {X 0,Y 237.042,Z 991.389,A -85,B 0,C 180,E1 3961.38,E2 3961.38} C_VEL
LIN {X 0,Y 256.976,Z 976.881,A -85,B 0,C 180,E1 3959.625,E2 3959.625} C_VEL
LIN {X 0,Y 269.29,Z 967.099,A -85,B 0,C 180,E1 3958.683,E2 3958.683} C_VEL
LIN {X 0,Y 257.988,Z 976.152,A -85,B 0,C 180,E1 3957.841,E2 3957.841} C_VEL
LIN {X 0,Y 251.867,Z 980.912,A -85,B 0,C 180,E1 3957.587,E2 3957.587} C_VEL
LIN {X 0,Y 234.477,Z 993.06,A -85,B 0,C 180,E1 3957.659,E2 3957.659} C_VEL
LIN {X 0,Y 228.997,Z 996.557,A -85,B 0,C 180,E1 3957.364,E2 3957.364} C_VEL
LIN {X 0,Y 209.643,Z 1008.405,A -85,B 0,C 180,E1 3955.429,E2 3955.429} C_VEL
LIN {X 0,Y 185.606,Z 1021.355,A -85,B 0,C 180,E1 3952.407,E2 3952.407} C_VEL
LIN {X 0,Y 164.99,Z 1030.981,A -85,B 0,C 180,E1 3949.042,E2 3949.042} C_VEL
LIN {X 0,Y 145.084,Z 1039.201,A -85,B 0,C 180,E1 3944.763,E2 3944.763} C_VEL
LIN {X 0,Y 122.093,Z 1047.354,A -85,B 0,C 180,E1 3937.732,E2 3937.732} C_VEL
LIN {X 0,Y 105.124,Z 1052.535,A -85,B 0,C 180,E1 3929.945,E2 3929.945} C_VEL
LIN {X 0,Y 90.008,Z 1056.666,A -85,B 0,C 180,E1 3919.048,E2 3919.048} C_VEL
LIN {X 0,Y 77.418,Z 1059.773,A -85,B 0,C 180,E1 3901.974,E2 3901.974} C_VEL
LIN {X 0,Y 72.663,Z 1060.924,A -85,B 0,C 180,E1 3885.975,E2 3885.975} C_VEL
LIN {X 0,Y 71.902,Z 1061.124,A -85,B 0,C 180,E1 3873.987,E2 3873.987} C_VEL
LIN {X 0,Y 71.906,Z 1060.876,A -85,B 0,C 180,E1 3865.214,E2 3865.214} C_VEL
LIN {X 0,Y 72.892,Z 1059.939,A -85,B 0,C 180,E1 3852.436,E2 3852.436} C_VEL
LIN {X 0,Y 78.76,Z 1057.548,A -85,B 0,C 180,E1 3835.16,E2 3835.16} C_VEL
LIN {X 0,Y 91.485,Z 1053.101,A -85,B 0,C 180,E1 3819.34,E2 3819.34} C_VEL
LIN {X 0,Y 105.636,Z 1048.155,A -85,B 0,C 180,E1 3809.447,E2 3809.447} C_VEL
LIN {X 0,Y 124.298,Z 1041.145,A -85,B 0,C 180,E1 3801.072,E2 3801.072} C_VEL
LIN {X 0,Y 145.72,Z 1031.899,A -85,B 0,C 180,E1 3794.65,E2 3794.65} C_VEL
LIN {X 0,Y 163.827,Z 1023.154,A -85,B 0,C 180,E1 3790.695,E2 3790.695} C_VEL
LIN {X 0,Y 185.397,Z 1011.538,A -85,B 0,C 180,E1 3787.093,E2 3787.093} C_VEL
LIN {X 0,Y 206.568,Z 998.388,A -85,B 0,C 180,E1 3784.34,E2 3784.34} C_VEL
LIN {X 0,Y 224.182,Z 986.233,A -85,B 0,C 180,E1 3782.472,E2 3782.472} C_VEL
LIN {X 0,Y 244.986,Z 970.271,A -85,B 0,C 180,E1 3780.635,E2 3780.635} C_VEL
LIN {X 0,Y 263.993,Z 953.582,A -85,B 0,C 180,E1 3779.219,E2 3779.219} C_VEL
LIN {X 0,Y 278.091,Z 939.934,A -85,B 0,C 180,E1 3778.291,E2 3778.291} C_VEL
LIN {X 0,Y 261.093,Z 956.22,A -85,B 0,C 180,E1 3777.146,E2 3777.146} C_VEL
LIN {X 0,Y 240.697,Z 973.5,A -85,B 0,C 180,E1 3775.552,E2 3775.552} C_VEL
LIN {X 0,Y 223.219,Z 986.694,A -85,B 0,C 180,E1 3773.945,E2 3773.945} C_VEL
LIN {X 0,Y 204.992,Z 999.116,A -85,B 0,C 180,E1 3771.958,E2 3771.958} C_VEL
LIN {X 0,Y 181.458,Z 1013.268,A -85,B 0,C 180,E1 3768.762,E2 3768.762} C_VEL
LIN {X 0,Y 163.118,Z 1022.977,A -85,B 0,C 180,E1 3765.582,E2 3765.582} C_VEL
LIN {X 0,Y 144.506,Z 1031.823,A -85,B 0,C 180,E1 3761.432,E2 3761.432} C_VEL
LIN {X 0,Y 121.969,Z 1041.233,A -85,B 0,C 180,E1 3754.39,E2 3754.39} C_VEL
LIN {X 0,Y 105.328,Z 1047.364,A -85,B 0,C 180,E1 3746.656,E2 3746.656} C_VEL
LIN {X 0,Y 91.026,Z 1052.25,A -85,B 0,C 180,E1 3736.467,E2 3736.467} C_VEL
LIN {X 0,Y 78.231,Z 1056.542,A -85,B 0,C 180,E1 3719.898,E2 3719.898} C_VEL
LIN {X 0,Y 73.053,Z 1058.594,A -85,B 0,C 180,E1 3704.262,E2 3704.262} C_VEL
LIN {X 0,Y 71.95,Z 1059.505,A -85,B 0,C 180,E1 3690.796,E2 3690.796} C_VEL
LIN {X 0,Y 72.002,Z 1059.805,A -85,B 0,C 180,E1 3680.394,E2 3680.394} C_VEL
LIN {X 0,Y 74.498,Z 1059.269,A -85,B 0,C 180,E1 3663.71,E2 3663.71} C_VEL
LIN {X 0,Y 82.499,Z 1057.417,A -85,B 0,C 180,E1 3647.256,E2 3647.256} C_VEL
LIN {X 0,Y 94.447,Z 1054.522,A -85,B 0,C 180,E1 3634.868,E2 3634.868} C_VEL
LIN {X 0,Y 112.626,Z 1049.621,A -85,B 0,C 180,E1 3623.876,E2 3623.876} C_VEL
LIN {X 0,Y 133.205,Z 1042.914,A -85,B 0,C 180,E1 3616.092,E2 3616.092} C_VEL
LIN {X 0,Y 151.871,Z 1035.994,A -85,B 0,C 180,E1 3611.191,E2 3611.191} C_VEL
LIN {X 0,Y 175.177,Z 1026.054,A -85,B 0,C 180,E1 3606.7,E2 3606.7} C_VEL
LIN {X 0,Y 196.368,Z 1015.509,A -85,B 0,C 180,E1 3603.615,E2 3603.615} C_VEL
LIN {X 0,Y 216.145,Z 1004.445,A -85,B 0,C 180,E1 3601.325,E2 3601.325} C_VEL
LIN {X 0,Y 240.002,Z 989.202,A -85,B 0,C 180,E1 3599.096,E2 3599.096} C_VEL
LIN {X 0,Y 244.802,Z 985.846,A -85,B 0,C 180,E1 3598.706,E2 3598.706} C_VEL
LIN {X 0,Y 228.997,Z 996.557,A -85,B 0,C 180,E1 3597.364,E2 3597.364} C_VEL
LIN {X 0,Y 222.522,Z 1000.718,A -85,B 0,C 180,E1 3597.025,E2 3597.025} C_VEL
LIN {X 0,Y 204.148,Z 1011.355,A -85,B 0,C 180,E1 3596.965,E2 3596.965} C_VEL
LIN {X 0,Y 198.405,Z 1014.345,A -85,B 0,C 180,E1 3596.58,E2 3596.58} C_VEL
LIN {X 0,Y 178.896,Z 1024.124,A -85,B 0,C 180,E1 3594.199,E2 3594.199} C_VEL
LIN {X 0,Y 156.082,Z 1034.228,A -85,B 0,C 180,E1 3590.591,E2 3590.591} C_VEL
LIN {X 0,Y 133.174,Z 1042.73,A -85,B 0,C 180,E1 3585.592,E2 3585.592} C_VEL
LIN {X 0,Y 114.117,Z 1048.861,A -85,B 0,C 180,E1 3579.64,E2 3579.64} C_VEL
LIN {X 0,Y 93.728,Z 1054.518,A -85,B 0,C 180,E1 3569.78,E2 3569.78} C_VEL
LIN {X 0,Y 77.678,Z 1058.186,A -85,B 0,C 180,E1 3556.124,E2 3556.124} C_VEL
LIN {X 0,Y 68.435,Z 1060.128,A -85,B 0,C 180,E1 3540.756,E2 3540.756} C_VEL
LIN {X 0,Y 64.417,Z 1060.947,A -85,B 0,C 180,E1 3524.381,E2 3524.381} C_VEL
LIN {X 0,Y 63.903,Z 1060.997,A -85,B 0,C 180,E1 3512.691,E2 3512.691} C_VEL
LIN {X 0,Y 63.984,Z 1060.723,A -85,B 0,C 180,E1 3501.915,E2 3501.915} C_VEL
LIN {X 0,Y 66.908,Z 1059.188,A -85,B 0,C 180,E1 3483.364,E2 3483.364} C_VEL
LIN {X 0,Y 75.97,Z 1056.189,A -85,B 0,C 180,E1 3465.769,E2 3465.769} C_VEL
LIN {X 0,Y 88.633,Z 1052.295,A -85,B 0,C 180,E1 3453.405,E2 3453.405} C_VEL
LIN {X 0,Y 106.541,Z 1046.466,A -85,B 0,C 180,E1 3443.115,E2 3443.115} C_VEL
LIN {X 0,Y 128.129,Z 1038.342,A -85,B 0,C 180,E1 3435.387,E2 3435.387} C_VEL
LIN {X 0,Y 146.589,Z 1030.495,A -85,B 0,C 180,E1 3430.821,E2 3430.821} C_VEL
LIN {X 0,Y 169.141,Z 1019.698,A -85,B 0,C 180,E1 3426.716,E2 3426.716} C_VEL
LIN {X 0,Y 190.393,Z 1007.857,A -85,B 0,C 180,E1 3423.789,E2 3423.789} C_VEL
LIN {X 0,Y 209.071,Z 996.238,A -85,B 0,C 180,E1 3421.733,E2 3421.733} C_VEL
LIN {X 0,Y 229.973,Z 981.736,A -85,B 0,C 180,E1 3419.851,E2 3419.851} C_VEL
LIN {X 0,Y 250.075,Z 965.73,A -85,B 0,C 180,E1 3418.343,E2 3418.343} C_VEL
LIN {X 0,Y 250.835,Z 965.085,A -85,B 0,C 180,E1 3418.269,E2 3418.269} C_VEL
LIN {X 0,Y 231.181,Z 980.724,A -85,B 0,C 180,E1 3416.777,E2 3416.777} C_VEL
LIN {X 0,Y 209.395,Z 995.848,A -85,B 0,C 180,E1 3414.794,E2 3414.794} C_VEL
LIN {X 0,Y 190.525,Z 1007.514,A -85,B 0,C 180,E1 3412.693,E2 3412.693} C_VEL
LIN {X 0,Y 167.792,Z 1019.989,A -85,B 0,C 180,E1 3409.496,E2 3409.496} C_VEL
LIN {X 0,Y 146.611,Z 1029.995,A -85,B 0,C 180,E1 3405.566,E2 3405.566} C_VEL
LIN {X 0,Y 128.011,Z 1037.796,A -85,B 0,C 180,E1 3400.929,E2 3400.929} C_VEL
LIN {X 0,Y 106.471,Z 1045.748,A -85,B 0,C 180,E1 3393.145,E2 3393.145} C_VEL
LIN {X 0,Y 88.882,Z 1051.36,A -85,B 0,C 180,E1 3383.008,E2 3383.008} C_VEL
LIN {X 0,Y 75.859,Z 1055.26,A -85,B 0,C 180,E1 3370.23,E2 3370.23} C_VEL
LIN {X 0,Y 66.501,Z 1058.289,A -85,B 0,C 180,E1 3351.152,E2 3351.152} C_VEL
LIN {X 0,Y 63.982,Z 1059.521,A -85,B 0,C 180,E1 3333.583,E2 3333.583} C_VEL
LIN {X 0,Y 63.95,Z 1059.795,A -85,B 0,C 180,E1 3322.814,E2 3322.814} C_VEL
LIN {X 0,Y 65.395,Z 1059.619,A -85,B 0,C 180,E1 3307.527,E2 3307.527} C_VEL
LIN {X 0,Y 73.12,Z 1058.256,A -85,B 0,C 180,E1 3287.928,E2 3287.928} C_VEL
LIN {X 0,Y 87.509,Z 1055.121,A -85,B 0,C 180,E1 3272.271,E2 3272.271} C_VEL
LIN {X 0,Y 103.012,Z 1051.313,A -85,B 0,C 180,E1 3262.762,E2 3262.762} C_VEL
LIN {X 0,Y 124.003,Z 1045.336,A -85,B 0,C 180,E1 3254.622,E2 3254.622} C_VEL
LIN {X 0,Y 146.712,Z 1037.41,A -85,B 0,C 180,E1 3248.804,E2 3248.804} C_VEL
LIN {X 0,Y 166.649,Z 1029.404,A -85,B 0,C 180,E1 3245.131,E2 3245.131} C_VEL
LIN {X 0,Y 191.066,Z 1018.057,A -85,B 0,C 180,E1 3241.741,E2 3241.741} C_VEL
LIN {X 0,Y 211.984,Z 1006.765,A -85,B 0,C 180,E1 3239.489,E2 3239.489} C_VEL
LIN {X 0,Y 220.127,Z 1002.101,A -85,B 0,C 180,E1 3238.699,E2 3238.699} C_VEL
LIN {X 0,Y 198.405,Z 1014.345,A -85,B 0,C 180,E1 3236.58,E2 3236.58} C_VEL
LIN {X 0,Y 191.629,Z 1017.888,A -85,B 0,C 180,E1 3236.13,E2 3236.13} C_VEL
LIN {X 0,Y 172.418,Z 1026.895,A -85,B 0,C 180,E1 3235.874,E2 3235.874} C_VEL
LIN {X 0,Y 166.47,Z 1029.399,A -85,B 0,C 180,E1 3235.351,E2 3235.351} C_VEL
LIN {X 0,Y 146.184,Z 1037.487,A -85,B 0,C 180,E1 3232.137,E2 3232.137} C_VEL
LIN {X 0,Y 124.718,Z 1044.91,A -85,B 0,C 180,E1 3227.498,E2 3227.498} C_VEL
LIN {X 0,Y 100.899,Z 1051.705,A -85,B 0,C 180,E1 3219.706,E2 3219.706} C_VEL
LIN {X 0,Y 83.761,Z 1055.764,A -85,B 0,C 180,E1 3210.626,E2 3210.626} C_VEL
LIN {X 0,Y 68.683,Z 1058.823,A -85,B 0,C 180,E1 3196.711,E2 3196.711} C_VEL
LIN {X 0,Y 58.08,Z 1060.677,A -85,B 0,C 180,E1 3174.405,E2 3174.405} C_VEL
LIN {X 0,Y 55.924,Z 1060.98,A -85,B 0,C 180,E1 3156.159,E2 3156.159} C_VEL
LIN {X 0,Y 55.9,Z 1060.757,A -85,B 0,C 180,E1 3145.898,E2 3145.898} C_VEL
LIN {X 0,Y 56.871,Z 1060.032,A -85,B 0,C 180,E1 3131.551,E2 3131.551} C_VEL
LIN {X 0,Y 62.269,Z 1058.272,A -85,B 0,C 180,E1 3113.55,E2 3113.55} C_VEL
LIN {X 0,Y 73.328,Z 1055.26,A -85,B 0,C 180,E1 3097.733,E2 3097.733} C_VEL
LIN {X 0,Y 92.829,Z 1049.695,A -85,B 0,C 180,E1 3083.716,E2 3083.716} C_VEL
LIN {X 0,Y 112.2,Z 1043.316,A -85,B 0,C 180,E1 3075.75,E2 3075.75} C_VEL
LIN {X 0,Y 132.112,Z 1035.869,A -85,B 0,C 180,E1 3070.296,E2 3070.296} C_VEL
LIN {X 0,Y 156.731,Z 1025.118,A -85,B 0,C 180,E1 3065.605,E2 3065.605} C_VEL
LIN {X 0,Y 176.199,Z 1015.33,A -85,B 0,C 180,E1 3062.864,E2 3062.864} C_VEL
LIN {X 0,Y 196.986,Z 1003.582,A -85,B 0,C 180,E1 3060.561,E2 3060.561} C_VEL
LIN {X 0,Y 220.046,Z 988.604,A -85,B 0,C 180,E1 3058.529,E2 3058.529} C_VEL
LIN {X 0,Y 223.551,Z 986.138,A -85,B 0,C 180,E1 3058.26,E2 3058.26} C_VEL
LIN {X 0,Y 205.314,Z 998.298,A -85,B 0,C 180,E1 3056.712,E2 3056.712} C_VEL
LIN {X 0,Y 182.558,Z 1011.778,A -85,B 0,C 180,E1 3054.342,E2 3054.342} C_VEL
LIN {X 0,Y 160.61,Z 1022.964,A -85,B 0,C 180,E1 3051.407,E2 3051.407} C_VEL
LIN {X 0,Y 141.072,Z 1031.761,A -85,B 0,C 180,E1 3047.988,E2 3047.988} C_VEL
LIN {X 0,Y 116.703,Z 1041.227,A -85,B 0,C 180,E1 3041.993,E2 3041.993} C_VEL
LIN {X 0,Y 98.101,Z 1047.385,A -85,B 0,C 180,E1 3035.109,E2 3035.109} C_VEL
LIN {X 0,Y 81.358,Z 1052.296,A -85,B 0,C 180,E1 3025.428,E2 3025.428} C_VEL
LIN {X 0,Y 65.143,Z 1056.639,A -85,B 0,C 180,E1 3007.876,E2 3007.876} C_VEL
LIN {X 0,Y 57.591,Z 1058.78,A -85,B 0,C 180,E1 2988.21,E2 2988.21} C_VEL
LIN {X 0,Y 55.952,Z 1059.648,A -85,B 0,C 180,E1 2972.048,E2 2972.048} C_VEL
LIN {X 0,Y 56.018,Z 1059.926,A -85,B 0,C 180,E1 2959.717,E2 2959.717} C_VEL
LIN {X 0,Y 59.297,Z 1059.576,A -85,B 0,C 180,E1 2939.316,E2 2939.316} C_VEL
LIN {X 0,Y 70.56,Z 1057.64,A -85,B 0,C 180,E1 2918.795,E2 2918.795} C_VEL
LIN {X 0,Y 85.586,Z 1054.692,A -85,B 0,C 180,E1 2905.897,E2 2905.897} C_VEL
LIN {X 0,Y 106.263,Z 1049.856,A -85,B 0,C 180,E1 2895.836,E2 2895.836} C_VEL
LIN {X 0,Y 128.614,Z 1043.244,A -85,B 0,C 180,E1 2889.127,E2 2889.127} C_VEL
LIN {X 0,Y 148.549,Z 1036.353,A -85,B 0,C 180,E1 2885.002,E2 2885.002} C_VEL
LIN {X 0,Y 172.034,Z 1026.932,A -85,B 0,C 180,E1 2881.431,E2 2881.431} C_VEL
LIN {X 0,Y 195.021,Z 1015.958,A -85,B 0,C 180,E1 2878.798,E2 2878.798} C_VEL
LIN {X 0,Y 195.58,Z 1015.671,A -85,B 0,C 180,E1 2878.742,E2 2878.742} C_VEL
LIN {X 0,Y 173.351,Z 1026.435,A -85,B 0,C 180,E1 2876.255,E2 2876.255} C_VEL
LIN {X 0,Y 166.47,Z 1029.399,A -85,B 0,C 180,E1 2875.351,E2 2875.351} C_VEL
LIN {X 0,Y 159.469,Z 1032.298,A -85,B 0,C 180,E1 2874.724,E2 2874.724} C_VEL
LIN {X 0,Y 139.595,Z 1039.616,A -85,B 0,C 180,E1 2874.126,E2 2874.126} C_VEL
LIN {X 0,Y 133.499,Z 1041.599,A -85,B 0,C 180,E1 2873.381,E2 2873.381} C_VEL
LIN {X 0,Y 112.2,Z 1048.044,A -85,B 0,C 180,E1 2868.603,E2 2868.603} C_VEL
LIN {X 0,Y 91.655,Z 1053.26,A -85,B 0,C 180,E1 2861.643,E2 2861.643} C_VEL
LIN {X 0,Y 69.401,Z 1057.727,A -85,B 0,C 180,E1 2848.216,E2 2848.216} C_VEL
LIN {X 0,Y 55.888,Z 1059.865,A -85,B 0,C 180,E1 2831.286,E2 2831.286} C_VEL
LIN {X 0,Y 49.259,Z 1060.75,A -85,B 0,C 180,E1 2811.431,E2 2811.431} C_VEL
LIN {X 0,Y 47.904,Z 1060.854,A -85,B 0,C 180,E1 2794.79,E2 2794.79} C_VEL
LIN {X 0,Y 47.917,Z 1060.651,A -85,B 0,C 180,E1 2784.012,E2 2784.012} C_VEL
LIN {X 0,Y 50.302,Z 1059.625,A -85,B 0,C 180,E1 2763.445,E2 2763.445} C_VEL
LIN {X 0,Y 61.359,Z 1056.938,A -85,B 0,C 180,E1 2740.014,E2 2740.014} C_VEL
LIN {X 0,Y 78.41,Z 1052.646,A -85,B 0,C 180,E1 2724.886,E2 2724.886} C_VEL
LIN {X 0,Y 95.855,Z 1047.746,A -85,B 0,C 180,E1 2716.328,E2 2716.328} C_VEL
LIN {X 0,Y 118.574,Z 1040.375,A -85,B 0,C 180,E1 2709.388,E2 2709.388} C_VEL
LIN {X 0,Y 141.473,Z 1031.388,A -85,B 0,C 180,E1 2704.768,E2 2704.768} C_VEL
LIN {X 0,Y 161.069,Z 1022.609,A -85,B 0,C 180,E1 2701.894,E2 2701.894} C_VEL
LIN {X 0,Y 184.994,Z 1010.35,A -85,B 0,C 180,E1 2699.236,E2 2699.236} C_VEL
LIN {X 0,Y 195.751,Z 1004.14,A -85,B 0,C 180,E1 2698.213,E2 2698.213} C_VEL
LIN {X 0,Y 175.361,Z 1015.37,A -85,B 0,C 180,E1 2696.217,E2 2696.217} C_VEL
LIN {X 0,Y 154.923,Z 1025.328,A -85,B 0,C 180,E1 2693.682,E2 2693.682} C_VEL
LIN {X 0,Y 130.155,Z 1035.674,A -85,B 0,C 180,E1 2689.522,E2 2689.522} C_VEL
LIN {X 0,Y 109.906,Z 1042.866,A -85,B 0,C 180,E1 2684.653,E2 2684.653} C_VEL
LIN {X 0,Y 89.034,Z 1049.272,A -85,B 0,C 180,E1 2677.055,E2 2677.055} C_VEL
LIN {X 0,Y 68.972,Z 1054.391,A -85,B 0,C 180,E1 2664.274,E2 2664.274} C_VEL
LIN {X 0,Y 55.869,Z 1057.41,A -85,B 0,C 180,E1 2647.48,E2 2647.48} C_VEL
LIN {X 0,Y 49.313,Z 1059.076,A -85,B 0,C 180,E1 2627.636,E2 2627.636} C_VEL
LIN {X 0,Y 47.949,Z 1059.753,A -85,B 0,C 180,E1 2611.194,E2 2611.194} C_VEL
LIN {X 0,Y 48.092,Z 1060.014,A -85,B 0,C 180,E1 2597.742,E2 2597.742} C_VEL
LIN {X 0,Y 52.658,Z 1059.597,A -85,B 0,C 180,E1 2573.939,E2 2573.939} C_VEL
LIN {X 0,Y 65.656,Z 1057.696,A -85,B 0,C 180,E1 2553.112,E2 2553.112} C_VEL
LIN {X 0,Y 81.447,Z 1054.896,A -85,B 0,C 180,E1 2541.09,E2 2541.09} C_VEL
LIN {X 0,Y 103.146,Z 1050.151,A -85,B 0,C 180,E1 2531.74,E2 2531.74} C_VEL
LIN {X 0,Y 126.586,Z 1043.561,A -85,B 0,C 180,E1 2525.583,E2 2525.583} C_VEL
LIN {X 0,Y 147.064,Z 1036.709,A -85,B 0,C 180,E1 2521.896,E2 2521.896} C_VEL
LIN {X 0,Y 170.745,Z 1027.469,A -85,B 0,C 180,E1 2518.767,E2 2518.767} C_VEL
LIN {X 0,Y 147.395,Z 1036.715,A -85,B 0,C 180,E1 2515.719,E2 2515.719} C_VEL
LIN {X 0,Y 133.499,Z 1041.599,A -85,B 0,C 180,E1 2513.381,E2 2513.381} C_VEL
LIN {X 0,Y 126.343,Z 1043.839,A -85,B 0,C 180,E1 2512.47,E2 2512.47} C_VEL
LIN {X 0,Y 106.001,Z 1049.417,A -85,B 0,C 180,E1 2511.221,E2 2511.221} C_VEL
LIN {X 0,Y 99.855,Z 1050.86,A -85,B 0,C 180,E1 2510.04,E2 2510.04} C_VEL
LIN {X 0,Y 78.577,Z 1055.376,A -85,B 0,C 180,E1 2502.218,E2 2502.218} C_VEL
LIN {X 0,Y 60.818,Z 1058.365,A -85,B 0,C 180,E1 2490.616,E2 2490.616} C_VEL
LIN {X 0,Y 45.42,Z 1060.419,A -85,B 0,C 180,E1 2468.054,E2 2468.054} C_VEL
LIN {X 0,Y 40.042,Z 1060.835,A -85,B 0,C 180,E1 2440.067,E2 2440.067} C_VEL
LIN {X 0,Y 39.898,Z 1060.637,A -85,B 0,C 180,E1 2427.128,E2 2427.128} C_VEL
LIN {X 0,Y 41.065,Z 1060.055,A -85,B 0,C 180,E1 2408.579,E2 2408.579} C_VEL
LIN {X 0,Y 48.335,Z 1058.412,A -85,B 0,C 180,E1 2385.305,E2 2385.305} C_VEL
